LIN {X 0,Y 497.703,Z 599.514,A -85,B 0,C 180,E1 23826.812,E2 23826.812} C_VEL
LIN {X 0,Y 498.495,Z 582.352,A -85,B 0,C 180,E1 23826.005,E2 23826.005} C_VEL
LIN {X 0,Y 499.076,Z 563.889,A -85,B 0,C 180,E1 23825.37,E2 23825.37} C_VEL
LIN {X 0,Y 499.352,Z 545.212,A -85,B 0,C 180,E1 23824.95,E2 23824.95} C_VEL
LIN {X 0,Y 500.791,Z 353.157,A -85,B 0,C 180,E1 23822.188,E2 23822.188} C_VEL
LIN {X 0,Y 497.596,Z 338.367,A -85,B 0,C 180,E1 23821.709,E2 23821.709} C_VEL
LIN {X 0,Y 497.97,Z 328.618,A -85,B 0,C 180,E1 23820.732,E2 23820.732} C_VEL
LIN {X 0,Y 491.564,Z 309.601,A -85,B 0,C 180,E1 23818.115,E2 23818.115} C_VEL
LIN {X 0,Y 488.836,Z 301.801,A -85,B 0,C 180,E1 23816.953,E2 23816.953} C_VEL
LIN {X 0,Y 488.821,Z 301.599,A -85,B 0,C 180,E1 23813.618,E2 23813.618} C_VEL
LIN {X 0,Y 488.832,Z 301.582,A -85,B 0,C 180,E1 23810.041,E2 23810.041} C_VEL
LIN {X 0,Y 488.806,Z 301.568,A -85,B 0,C 180,E1 23806.566,E2 23806.566} C_VEL
LIN {X 0,Y 488.795,Z 301.598,A -85,B 0,C 180,E1 23803.093,E2 23803.093} C_VEL
LIN {X 0,Y 488.83,Z 301.598,A -85,B 0,C 180,E1 23799.656,E2 23799.656} C_VEL
LIN {X 0,Y 488.827,Z 301.593,A -85,B 0,C 180,E1 23796.092,E2 23796.092} C_VEL
LIN {X 0,Y 488.788,Z 301.595,A -85,B 0,C 180,E1 23792.568,E2 23792.568} C_VEL
LIN {X 0,Y 488.784,Z 301.593,A -85,B 0,C 180,E1 23789,E2 23789} C_VEL
LIN {X 0,Y 488.822,Z 301.587,A -85,B 0,C 180,E1 23785.569,E2 23785.569} C_VEL
LIN {X 0,Y 488.805,Z 301.596,A -85,B 0,C 180,E1 23782.09,E2 23782.09} C_VEL
LIN {X 0,Y 488.769,Z 301.592,A -85,B 0,C 180,E1 23778.61,E2 23778.61} C_VEL
LIN {X 0,Y 488.776,Z 301.588,A -85,B 0,C 180,E1 23775.058,E2 23775.058} C_VEL
LIN {X 0,Y 488.818,Z 301.596,A -85,B 0,C 180,E1 23771.684,E2 23771.684} C_VEL
LIN {X 0,Y 488.765,Z 301.585,A -85,B 0,C 180,E1 23768.233,E2 23768.233} C_VEL
LIN {X 0,Y 488.755,Z 301.597,A -85,B 0,C 180,E1 23764.694,E2 23764.694} C_VEL
LIN {X 0,Y 488.797,Z 301.596,A -85,B 0,C 180,E1 23761.29,E2 23761.29} C_VEL
LIN {X 0,Y 488.775,Z 301.592,A -85,B 0,C 180,E1 23757.89,E2 23757.89} C_VEL
LIN {X 0,Y 488.754,Z 301.599,A -85,B 0,C 180,E1 23754.483,E2 23754.483} C_VEL
LIN {X 0,Y 488.789,Z 301.592,A -85,B 0,C 180,E1 23751.057,E2 23751.057} C_VEL
LIN {X 0,Y 488.805,Z 301.592,A -85,B 0,C 180,E1 23747.598,E2 23747.598} C_VEL
LIN {X 0,Y 488.767,Z 301.599,A -85,B 0,C 180,E1 23744.212,E2 23744.212} C_VEL
LIN {X 0,Y 488.78,Z 301.595,A -85,B 0,C 180,E1 23740.647,E2 23740.647} C_VEL
LIN {X 0,Y 488.836,Z 301.585,A -85,B 0,C 180,E1 23737.258,E2 23737.258} C_VEL
LIN {X 0,Y 488.792,Z 301.599,A -85,B 0,C 180,E1 23733.779,E2 23733.779} C_VEL
LIN {X 0,Y 488.782,Z 301.597,A -85,B 0,C 180,E1 23730.328,E2 23730.328} C_VEL
LIN {X 0,Y 488.822,Z 301.594,A -85,B 0,C 180,E1 23726.898,E2 23726.898} C_VEL
LIN {X 0,Y 488.826,Z 301.564,A -85,B 0,C 180,E1 23723.301,E2 23723.301} C_VEL
LIN {X 0,Y 488.793,Z 301.59,A -85,B 0,C 180,E1 23719.883,E2 23719.883} C_VEL
LIN {X 0,Y 488.796,Z 301.598,A -85,B 0,C 180,E1 23716.225,E2 23716.225} C_VEL
LIN {X 0,Y 488.826,Z 301.575,A -85,B 0,C 180,E1 23712.751,E2 23712.751} C_VEL
LIN {X 0,Y 488.839,Z 301.65,A -85,B 0,C 180,E1 23711.1,E2 23711.1} C_VEL
LIN {X 0,Y 489.193,Z 303.151,A -85,B 0,C 180,E1 23710.866,E2 23710.866} C_VEL
LIN {X 0,Y 497.247,Z 321.838,A -85,B 0,C 180,E1 23708.815,E2 23708.815} C_VEL
LIN {X 0,Y 502.538,Z 335.639,A -85,B 0,C 180,E1 23707.431,E2 23707.431} C_VEL
LIN {X 0,Y 500.242,Z 388.267,A -85,B 0,C 180,E1 23704.007,E2 23704.007} C_VEL
LIN {X 0,Y 502.743,Z 409.204,A -85,B 0,C 180,E1 23703.487,E2 23703.487} C_VEL
LIN {X 0,Y 499.827,Z 627.706,A -85,B 0,C 180,E1 23700.075,E2 23700.075} C_VEL
LIN {X 0,Y 499.277,Z 655.552,A -85,B 0,C 180,E1 23699.579,E2 23699.579} C_VEL
LIN {X 0,Y 498.434,Z 677.22,A -85,B 0,C 180,E1 23698.977,E2 23698.977} C_VEL
LIN {X 0,Y 497.483,Z 697.861,A -85,B 0,C 180,E1 23698.184,E2 23698.184} C_VEL
LIN {X 0,Y 496.413,Z 717.588,A -85,B 0,C 180,E1 23697.207,E2 23697.207} C_VEL
LIN {X 0,Y 495.194,Z 737.474,A -85,B 0,C 180,E1 23695.985,E2 23695.985} C_VEL
LIN {X 0,Y 493.989,Z 756.462,A -85,B 0,C 180,E1 23694.565,E2 23694.565} C_VEL
LIN {X 0,Y 492.797,Z 774.049,A -85,B 0,C 180,E1 23692.989,E2 23692.989} C_VEL
LIN {X 0,Y 491.739,Z 789.65,A -85,B 0,C 180,E1 23691.343,E2 23691.343} C_VEL
LIN {X 0,Y 490.759,Z 804.438,A -85,B 0,C 180,E1 23689.519,E2 23689.519} C_VEL
LIN {X 0,Y 490.048,Z 815.118,A -85,B 0,C 180,E1 23687.944,E2 23687.944} C_VEL
LIN {X 0,Y 489.28,Z 826.646,A -85,B 0,C 180,E1 23685.892,E2 23685.892} C_VEL
LIN {X 0,Y 488.709,Z 836.846,A -85,B 0,C 180,E1 23683.728,E2 23683.728} C_VEL
LIN {X 0,Y 488.31,Z 845.655,A -85,B 0,C 180,E1 23681.456,E2 23681.456} C_VEL
LIN {X 0,Y 488.088,Z 852.685,A -85,B 0,C 180,E1 23679.194,E2 23679.194} C_VEL
LIN {X 0,Y 487.97,Z 858.26,A -85,B 0,C 180,E1 23676.825,E2 23676.825} C_VEL
LIN {X 0,Y 487.913,Z 862.087,A -85,B 0,C 180,E1 23674.466,E2 23674.466} C_VEL
LIN {X 0,Y 487.908,Z 864.304,A -85,B 0,C 180,E1 23672.114,E2 23672.114} C_VEL
LIN {X 0,Y 487.906,Z 864.962,A -85,B 0,C 180,E1 23669.765,E2 23669.765} C_VEL
LIN {X 0,Y 487.905,Z 864.03,A -85,B 0,C 180,E1 23667.416,E2 23667.416} C_VEL
LIN {X 0,Y 487.929,Z 861.446,A -85,B 0,C 180,E1 23665.063,E2 23665.063} C_VEL
LIN {X 0,Y 487.987,Z 857.244,A -85,B 0,C 180,E1 23662.702,E2 23662.702} C_VEL
LIN {X 0,Y 488.126,Z 851.326,A -85,B 0,C 180,E1 23660.331,E2 23660.331} C_VEL
LIN {X 0,Y 488.381,Z 844.01,A -85,B 0,C 180,E1 23658.067,E2 23658.067} C_VEL
LIN {X 0,Y 488.823,Z 834.789,A -85,B 0,C 180,E1 23655.792,E2 23655.792} C_VEL
LIN {X 0,Y 489.44,Z 824.106,A -85,B 0,C 180,E1 23653.626,E2 23653.626} C_VEL
LIN {X 0,Y 490.253,Z 812.019,A -85,B 0,C 180,E1 23651.572,E2 23651.572} C_VEL
LIN {X 0,Y 491.025,Z 800.468,A -85,B 0,C 180,E1 23649.954,E2 23649.954} C_VEL
LIN {X 0,Y 492.085,Z 784.784,A -85,B 0,C 180,E1 23648.109,E2 23648.109} C_VEL
LIN {X 0,Y 493.241,Z 767.415,A -85,B 0,C 180,E1 23646.385,E2 23646.385} C_VEL
LIN {X 0,Y 494.4,Z 750.145,A -85,B 0,C 180,E1 23644.94,E2 23644.94} C_VEL
LIN {X 0,Y 495.552,Z 731.825,A -85,B 0,C 180,E1 23643.649,E2 23643.649} C_VEL
LIN {X 0,Y 496.728,Z 711.811,A -85,B 0,C 180,E1 23642.487,E2 23642.487} C_VEL
LIN {X 0,Y 497.765,Z 692.146,A -85,B 0,C 180,E1 23641.572,E2 23641.572} C_VEL
LIN {X 0,Y 498.696,Z 671.504,A -85,B 0,C 180,E1 23640.837,E2 23640.837} C_VEL
LIN {X 0,Y 499.453,Z 649.882,A -85,B 0,C 180,E1 23640.293,E2 23640.293} C_VEL
LIN {X 0,Y 502.656,Z 414.695,A -85,B 0,C 180,E1 23636.6,E2 23636.6} C_VEL
LIN {X 0,Y 502.523,Z 405.875,A -85,B 0,C 180,E1 23636.443,E2 23636.443} C_VEL
LIN {X 0,Y 500.189,Z 387.515,A -85,B 0,C 180,E1 23635.965,E2 23635.965} C_VEL
LIN {X 0,Y 502.552,Z 335.273,A -85,B 0,C 180,E1 23632.545,E2 23632.545} C_VEL
LIN {X 0,Y 494.184,Z 314.542,A -85,B 0,C 180,E1 23630.409,E2 23630.409} C_VEL
LIN {X 0,Y 488.897,Z 302.02,A -85,B 0,C 180,E1 23628.995,E2 23628.995} C_VEL
LIN {X 0,Y 488.827,Z 301.588,A -85,B 0,C 180,E1 23628.648,E2 23628.648} C_VEL
LIN {X 0,Y 488.832,Z 301.584,A -85,B 0,C 180,E1 23625.049,E2 23625.049} C_VEL
LIN {X 0,Y 488.802,Z 301.566,A -85,B 0,C 180,E1 23621.51,E2 23621.51} C_VEL
LIN {X 0,Y 488.79,Z 301.592,A -85,B 0,C 180,E1 23618.004,E2 23618.004} C_VEL
LIN {X 0,Y 488.813,Z 301.58,A -85,B 0,C 180,E1 23614.482,E2 23614.482} C_VEL
LIN {X 0,Y 488.834,Z 301.587,A -85,B 0,C 180,E1 23610.89,E2 23610.89} C_VEL
LIN {X 0,Y 488.79,Z 301.591,A -85,B 0,C 180,E1 23607.403,E2 23607.403} C_VEL
LIN {X 0,Y 488.779,Z 301.593,A -85,B 0,C 180,E1 23603.884,E2 23603.884} C_VEL
LIN {X 0,Y 488.816,Z 301.598,A -85,B 0,C 180,E1 23600.473,E2 23600.473} C_VEL
LIN {X 0,Y 488.801,Z 301.592,A -85,B 0,C 180,E1 23597.008,E2 23597.008} C_VEL
LIN {X 0,Y 488.765,Z 301.585,A -85,B 0,C 180,E1 23593.606,E2 23593.606} C_VEL
LIN {X 0,Y 488.783,Z 301.596,A -85,B 0,C 180,E1 23590.132,E2 23590.132} C_VEL
LIN {X 0,Y 488.827,Z 301.591,A -85,B 0,C 180,E1 23586.577,E2 23586.577} C_VEL
LIN {X 0,Y 488.77,Z 301.59,A -85,B 0,C 180,E1 23583.049,E2 23583.049} C_VEL
LIN {X 0,Y 488.753,Z 301.6,A -85,B 0,C 180,E1 23579.648,E2 23579.648} C_VEL
LIN {X 0,Y 488.794,Z 301.59,A -85,B 0,C 180,E1 23576.247,E2 23576.247} C_VEL
LIN {X 0,Y 488.783,Z 301.599,A -85,B 0,C 180,E1 23572.79,E2 23572.79} C_VEL
LIN {X 0,Y 488.756,Z 301.598,A -85,B 0,C 180,E1 23569.39,E2 23569.39} C_VEL
LIN {X 0,Y 488.783,Z 301.585,A -85,B 0,C 180,E1 23565.911,E2 23565.911} C_VEL
LIN {X 0,Y 488.808,Z 301.6,A -85,B 0,C 180,E1 23562.501,E2 23562.501} C_VEL
LIN {X 0,Y 488.771,Z 301.593,A -85,B 0,C 180,E1 23559.023,E2 23559.023} C_VEL
LIN {X 0,Y 488.775,Z 301.586,A -85,B 0,C 180,E1 23555.464,E2 23555.464} C_VEL
LIN {X 0,Y 488.83,Z 301.592,A -85,B 0,C 180,E1 23552.069,E2 23552.069} C_VEL
LIN {X 0,Y 488.806,Z 301.597,A -85,B 0,C 180,E1 23548.534,E2 23548.534} C_VEL
LIN {X 0,Y 488.781,Z 301.595,A -85,B 0,C 180,E1 23545.056,E2 23545.056} C_VEL
LIN {X 0,Y 488.801,Z 301.594,A -85,B 0,C 180,E1 23541.549,E2 23541.549} C_VEL
LIN {X 0,Y 488.832,Z 301.59,A -85,B 0,C 180,E1 23538.022,E2 23538.022} C_VEL
LIN {X 0,Y 488.81,Z 301.571,A -85,B 0,C 180,E1 23534.448,E2 23534.448} C_VEL
LIN {X 0,Y 488.793,Z 301.6,A -85,B 0,C 180,E1 23530.887,E2 23530.887} C_VEL
LIN {X 0,Y 488.804,Z 301.585,A -85,B 0,C 180,E1 23527.277,E2 23527.277} C_VEL
LIN {X 0,Y 488.829,Z 301.571,A -85,B 0,C 180,E1 23523.803,E2 23523.803} C_VEL
LIN {X 0,Y 488.825,Z 301.575,A -85,B 0,C 180,E1 23523.535,E2 23523.535} C_VEL
LIN {X 0,Y 488.707,Z 302.659,A -85,B 0,C 180,E1 23523.028,E2 23523.028} C_VEL
LIN {X 0,Y 488.366,Z 306.029,A -85,B 0,C 180,E1 23522.479,E2 23522.479} C_VEL
LIN {X 0,Y 487.643,Z 319.511,A -85,B 0,C 180,E1 23521.022,E2 23521.022} C_VEL
LIN {X 0,Y 488.549,Z 324.711,A -85,B 0,C 180,E1 23520.361,E2 23520.361} C_VEL
LIN {X 0,Y 490.865,Z 331.872,A -85,B 0,C 180,E1 23519.399,E2 23519.399} C_VEL
LIN {X 0,Y 490.606,Z 339.583,A -85,B 0,C 180,E1 23518.658,E2 23518.658} C_VEL
LIN {X 0,Y 494.065,Z 356.306,A -85,B 0,C 180,E1 23518.141,E2 23518.141} C_VEL
LIN {X 0,Y 492.291,Z 551.901,A -85,B 0,C 180,E1 23515.29,E2 23515.29} C_VEL
LIN {X 0,Y 491.896,Z 570.892,A -85,B 0,C 180,E1 23514.786,E2 23514.786} C_VEL
LIN {X 0,Y 491.192,Z 588.904,A -85,B 0,C 180,E1 23514.087,E2 23514.087} C_VEL
LIN {X 0,Y 490.248,Z 606.351,A -85,B 0,C 180,E1 23513.179,E2 23513.179} C_VEL
LIN {X 0,Y 489.098,Z 622.756,A -85,B 0,C 180,E1 23512.095,E2 23512.095} C_VEL
LIN {X 0,Y 487.851,Z 638.101,A -85,B 0,C 180,E1 23510.839,E2 23510.839} C_VEL
LIN {X 0,Y 486.5,Z 652.717,A -85,B 0,C 180,E1 23509.379,E2 23509.379} C_VEL
LIN {X 0,Y 485.184,Z 666.107,A -85,B 0,C 180,E1 23507.757,E2 23507.757} C_VEL
LIN {X 0,Y 483.924,Z 678.429,A -85,B 0,C 180,E1 23505.949,E2 23505.949} C_VEL
LIN {X 0,Y 482.864,Z 689.222,A -85,B 0,C 180,E1 23504.02,E2 23504.02} C_VEL
LIN {X 0,Y 481.974,Z 698.544,A -85,B 0,C 180,E1 23501.973,E2 23501.973} C_VEL
LIN {X 0,Y 481.314,Z 706.381,A -85,B 0,C 180,E1 23499.807,E2 23499.807} C_VEL
LIN {X 0,Y 480.863,Z 712.699,A -85,B 0,C 180,E1 23497.527,E2 23497.527} C_VEL
LIN {X 0,Y 480.577,Z 717.234,A -85,B 0,C 180,E1 23495.252,E2 23495.252} C_VEL
LIN {X 0,Y 480.428,Z 720.208,A -85,B 0,C 180,E1 23492.863,E2 23492.863} C_VEL
LIN {X 0,Y 480.381,Z 721.437,A -85,B 0,C 180,E1 23490.477,E2 23490.477} C_VEL
LIN {X 0,Y 480.403,Z 720.959,A -85,B 0,C 180,E1 23488.092,E2 23488.092} C_VEL
LIN {X 0,Y 480.492,Z 718.906,A -85,B 0,C 180,E1 23485.824,E2 23485.824} C_VEL
LIN {X 0,Y 480.694,Z 715.237,A -85,B 0,C 180,E1 23483.551,E2 23483.551} C_VEL
LIN {X 0,Y 481.06,Z 709.851,A -85,B 0,C 180,E1 23481.273,E2 23481.273} C_VEL
LIN {X 0,Y 481.58,Z 703.016,A -85,B 0,C 180,E1 23479.11,E2 23479.11} C_VEL
LIN {X 0,Y 482.32,Z 694.791,A -85,B 0,C 180,E1 23477.063,E2 23477.063} C_VEL
LIN {X 0,Y 483.286,Z 684.793,A -85,B 0,C 180,E1 23475.054,E2 23475.054} C_VEL
LIN {X 0,Y 484.416,Z 673.543,A -85,B 0,C 180,E1 23473.204,E2 23473.204} C_VEL
LIN {X 0,Y 485.68,Z 661.12,A -85,B 0,C 180,E1 23471.517,E2 23471.517} C_VEL
LIN {X 0,Y 487.013,Z 647.199,A -85,B 0,C 180,E1 23469.95,E2 23469.95} C_VEL
LIN {X 0,Y 488.338,Z 632.237,A -85,B 0,C 180,E1 23468.564,E2 23468.564} C_VEL
LIN {X 0,Y 489.56,Z 616.352,A -85,B 0,C 180,E1 23467.364,E2 23467.364} C_VEL
LIN {X 0,Y 490.6,Z 600.329,A -85,B 0,C 180,E1 23466.393,E2 23466.393} C_VEL
LIN {X 0,Y 491.444,Z 583.063,A -85,B 0,C 180,E1 23465.575,E2 23465.575} C_VEL
LIN {X 0,Y 492.049,Z 564.71,A -85,B 0,C 180,E1 23464.938,E2 23464.938} C_VEL
LIN {X 0,Y 492.337,Z 545.999,A -85,B 0,C 180,E1 23464.513,E2 23464.513} C_VEL
LIN {X 0,Y 493.96,Z 354.759,A -85,B 0,C 180,E1 23461.732,E2 23461.732} C_VEL
LIN {X 0,Y 490.529,Z 338.771,A -85,B 0,C 180,E1 23461.202,E2 23461.202} C_VEL
LIN {X 0,Y 490.727,Z 331.435,A -85,B 0,C 180,E1 23460.458,E2 23460.458} C_VEL
LIN {X 0,Y 484.023,Z 311.463,A -85,B 0,C 180,E1 23457.66,E2 23457.66} C_VEL
LIN {X 0,Y 480.917,Z 302.763,A -85,B 0,C 180,E1 23456.336,E2 23456.336} C_VEL
LIN {X 0,Y 480.867,Z 302.575,A -85,B 0,C 180,E1 23452.767,E2 23452.767} C_VEL
LIN {X 0,Y 480.863,Z 302.589,A -85,B 0,C 180,E1 23449.189,E2 23449.189} C_VEL
LIN {X 0,Y 480.883,Z 302.553,A -85,B 0,C 180,E1 23445.664,E2 23445.664} C_VEL
LIN {X 0,Y 480.895,Z 302.58,A -85,B 0,C 180,E1 23442.028,E2 23442.028} C_VEL
LIN {X 0,Y 480.867,Z 302.582,A -85,B 0,C 180,E1 23438.441,E2 23438.441} C_VEL
LIN {X 0,Y 480.848,Z 302.582,A -85,B 0,C 180,E1 23434.878,E2 23434.878} C_VEL
LIN {X 0,Y 480.86,Z 302.585,A -85,B 0,C 180,E1 23431.288,E2 23431.288} C_VEL
LIN {X 0,Y 480.894,Z 302.581,A -85,B 0,C 180,E1 23427.758,E2 23427.758} C_VEL
LIN {X 0,Y 480.86,Z 302.573,A -85,B 0,C 180,E1 23424.182,E2 23424.182} C_VEL
LIN {X 0,Y 480.835,Z 302.581,A -85,B 0,C 180,E1 23420.657,E2 23420.657} C_VEL
LIN {X 0,Y 480.84,Z 302.588,A -85,B 0,C 180,E1 23417.05,E2 23417.05} C_VEL
LIN {X 0,Y 480.885,Z 302.571,A -85,B 0,C 180,E1 23413.589,E2 23413.589} C_VEL
LIN {X 0,Y 480.844,Z 302.586,A -85,B 0,C 180,E1 23410.06,E2 23410.06} C_VEL
LIN {X 0,Y 480.818,Z 302.588,A -85,B 0,C 180,E1 23406.568,E2 23406.568} C_VEL
LIN {X 0,Y 480.836,Z 302.574,A -85,B 0,C 180,E1 23403.099,E2 23403.099} C_VEL
LIN {X 0,Y 480.876,Z 302.585,A -85,B 0,C 180,E1 23399.524,E2 23399.524} C_VEL
LIN {X 0,Y 480.831,Z 302.58,A -85,B 0,C 180,E1 23395.946,E2 23395.946} C_VEL
LIN {X 0,Y 480.818,Z 302.579,A -85,B 0,C 180,E1 23392.472,E2 23392.472} C_VEL
LIN {X 0,Y 480.845,Z 302.587,A -85,B 0,C 180,E1 23388.943,E2 23388.943} C_VEL
LIN {X 0,Y 480.886,Z 302.576,A -85,B 0,C 180,E1 23385.429,E2 23385.429} C_VEL
LIN {X 0,Y 480.839,Z 302.581,A -85,B 0,C 180,E1 23381.951,E2 23381.951} C_VEL
LIN {X 0,Y 480.834,Z 302.586,A -85,B 0,C 180,E1 23378.353,E2 23378.353} C_VEL
LIN {X 0,Y 480.87,Z 302.585,A -85,B 0,C 180,E1 23374.902,E2 23374.902} C_VEL
LIN {X 0,Y 480.897,Z 302.584,A -85,B 0,C 180,E1 23371.296,E2 23371.296} C_VEL
LIN {X 0,Y 480.853,Z 302.585,A -85,B 0,C 180,E1 23367.808,E2 23367.808} C_VEL
LIN {X 0,Y 480.845,Z 302.554,A -85,B 0,C 180,E1 23364.187,E2 23364.187} C_VEL
LIN {X 0,Y 480.874,Z 302.584,A -85,B 0,C 180,E1 23360.642,E2 23360.642} C_VEL
LIN {X 0,Y 480.892,Z 302.564,A -85,B 0,C 180,E1 23357.041,E2 23357.041} C_VEL
LIN {X 0,Y 480.874,Z 302.557,A -85,B 0,C 180,E1 23353.477,E2 23353.477} C_VEL
LIN {X 0,Y 480.906,Z 302.863,A -85,B 0,C 180,E1 23351.68,E2 23351.68} C_VEL
LIN {X 0,Y 483.793,Z 309.643,A -85,B 0,C 180,E1 23350.851,E2 23350.851} C_VEL
LIN {X 0,Y 493.151,Z 332.06,A -85,B 0,C 180,E1 23348.407,E2 23348.407} C_VEL
LIN {X 0,Y 495.521,Z 338.509,A -85,B 0,C 180,E1 23347.762,E2 23347.762} C_VEL
LIN {X 0,Y 493.157,Z 387.828,A -85,B 0,C 180,E1 23344.503,E2 23344.503} C_VEL
LIN {X 0,Y 495.787,Z 410.337,A -85,B 0,C 180,E1 23343.929,E2 23343.929} C_VEL
LIN {X 0,Y 492.138,Z 649.298,A -85,B 0,C 180,E1 23340.091,E2 23340.091} C_VEL
LIN {X 0,Y 491.304,Z 671.237,A -85,B 0,C 180,E1 23339.525,E2 23339.525} C_VEL
LIN {X 0,Y 490.246,Z 692.612,A -85,B 0,C 180,E1 23338.74,E2 23338.74} C_VEL
LIN {X 0,Y 489.065,Z 713.265,A -85,B 0,C 180,E1 23337.746,E2 23337.746} C_VEL
LIN {X 0,Y 487.862,Z 732.316,A -85,B 0,C 180,E1 23336.602,E2 23336.602} C_VEL
LIN {X 0,Y 486.592,Z 751.078,A -85,B 0,C 180,E1 23335.237,E2 23335.237} C_VEL
LIN {X 0,Y 485.262,Z 769.522,A -85,B 0,C 180,E1 23333.625,E2 23333.625} C_VEL
LIN {X 0,Y 484.067,Z 786.361,A -85,B 0,C 180,E1 23331.874,E2 23331.874} C_VEL
LIN {X 0,Y 483.041,Z 800.956,A -85,B 0,C 180,E1 23330.096,E2 23330.096} C_VEL
LIN {X 0,Y 482.123,Z 814.745,A -85,B 0,C 180,E1 23328.124,E2 23328.124} C_VEL
LIN {X 0,Y 481.36,Z 827.01,A -85,B 0,C 180,E1 23326.037,E2 23326.037} C_VEL
LIN {X 0,Y 480.828,Z 836.331,A -85,B 0,C 180,E1 23324.081,E2 23324.081} C_VEL
LIN {X 0,Y 480.378,Z 845.25,A -85,B 0,C 180,E1 23321.769,E2 23321.769} C_VEL
LIN {X 0,Y 480.123,Z 852.375,A -85,B 0,C 180,E1 23319.469,E2 23319.469} C_VEL
LIN {X 0,Y 479.983,Z 858.006,A -85,B 0,C 180,E1 23317.059,E2 23317.059} C_VEL
LIN {X 0,Y 479.919,Z 861.926,A -85,B 0,C 180,E1 23314.66,E2 23314.66} C_VEL
LIN {X 0,Y 479.907,Z 864.303,A -85,B 0,C 180,E1 23312.149,E2 23312.149} C_VEL
LIN {X 0,Y 479.906,Z 864.962,A -85,B 0,C 180,E1 23309.761,E2 23309.761} C_VEL
LIN {X 0,Y 479.907,Z 864.03,A -85,B 0,C 180,E1 23307.373,E2 23307.373} C_VEL
LIN {X 0,Y 479.931,Z 861.445,A -85,B 0,C 180,E1 23304.98,E2 23304.98} C_VEL
LIN {X 0,Y 479.994,Z 857.159,A -85,B 0,C 180,E1 23302.54,E2 23302.54} C_VEL
LIN {X 0,Y 480.146,Z 851.326,A -85,B 0,C 180,E1 23300.168,E2 23300.168} C_VEL
LIN {X 0,Y 480.431,Z 844.009,A -85,B 0,C 180,E1 23297.866,E2 23297.866} C_VEL
LIN {X 0,Y 480.919,Z 834.786,A -85,B 0,C 180,E1 23295.553,E2 23295.553} C_VEL
LIN {X 0,Y 481.435,Z 825.653,A -85,B 0,C 180,E1 23293.718,E2 23293.718} C_VEL
LIN {X 0,Y 482.226,Z 813.101,A -85,B 0,C 180,E1 23291.63,E2 23291.63} C_VEL
LIN {X 0,Y 483.169,Z 799.084,A -85,B 0,C 180,E1 23289.657,E2 23289.657} C_VEL
LIN {X 0,Y 484.324,Z 782.977,A -85,B 0,C 180,E1 23287.741,E2 23287.741} C_VEL
LIN {X 0,Y 485.559,Z 765.638,A -85,B 0,C 180,E1 23286.004,E2 23286.004} C_VEL
LIN {X 0,Y 486.861,Z 747.174,A -85,B 0,C 180,E1 23284.452,E2 23284.452} C_VEL
LIN {X 0,Y 488.045,Z 729.442,A -85,B 0,C 180,E1 23283.211,E2 23283.211} C_VEL
LIN {X 0,Y 489.249,Z 710.207,A -85,B 0,C 180,E1 23282.096,E2 23282.096} C_VEL
LIN {X 0,Y 490.344,Z 690.339,A -85,B 0,C 180,E1 23281.169,E2 23281.169} C_VEL
LIN {X 0,Y 491.367,Z 669.669,A -85,B 0,C 180,E1 23280.429,E2 23280.429} C_VEL
LIN {X 0,Y 492.173,Z 648.273,A -85,B 0,C 180,E1 23279.887,E2 23279.887} C_VEL
LIN {X 0,Y 495.806,Z 409.537,A -85,B 0,C 180,E1 23276.057,E2 23276.057} C_VEL
LIN {X 0,Y 493.099,Z 386.873,A -85,B 0,C 180,E1 23275.46,E2 23275.46} C_VEL
LIN {X 0,Y 495.495,Z 338.18,A -85,B 0,C 180,E1 23272.214,E2 23272.214} C_VEL
LIN {X 0,Y 486.73,Z 316.473,A -85,B 0,C 180,E1 23269.925,E2 23269.925} C_VEL
LIN {X 0,Y 480.947,Z 303.081,A -85,B 0,C 180,E1 23268.366,E2 23268.366} C_VEL
LIN {X 0,Y 480.86,Z 302.587,A -85,B 0,C 180,E1 23268.107,E2 23268.107} C_VEL
LIN {X 0,Y 480.875,Z 302.584,A -85,B 0,C 180,E1 23264.483,E2 23264.483} C_VEL
LIN {X 0,Y 480.898,Z 302.556,A -85,B 0,C 180,E1 23260.818,E2 23260.818} C_VEL
LIN {X 0,Y 480.878,Z 302.561,A -85,B 0,C 180,E1 23257.22,E2 23257.22} C_VEL
LIN {X 0,Y 480.849,Z 302.585,A -85,B 0,C 180,E1 23253.724,E2 23253.724} C_VEL
LIN {X 0,Y 480.851,Z 302.589,A -85,B 0,C 180,E1 23250.074,E2 23250.074} C_VEL
LIN {X 0,Y 480.887,Z 302.578,A -85,B 0,C 180,E1 23246.616,E2 23246.616} C_VEL
LIN {X 0,Y 480.875,Z 302.576,A -85,B 0,C 180,E1 23243.01,E2 23243.01} C_VEL
LIN {X 0,Y 480.835,Z 302.584,A -85,B 0,C 180,E1 23239.559,E2 23239.559} C_VEL
LIN {X 0,Y 480.836,Z 302.588,A -85,B 0,C 180,E1 23235.931,E2 23235.931} C_VEL
LIN {X 0,Y 480.877,Z 302.576,A -85,B 0,C 180,E1 23232.488,E2 23232.488} C_VEL
LIN {X 0,Y 480.849,Z 302.58,A -85,B 0,C 180,E1 23228.972,E2 23228.972} C_VEL
LIN {X 0,Y 480.818,Z 302.589,A -85,B 0,C 180,E1 23225.489,E2 23225.489} C_VEL
LIN {X 0,Y 480.827,Z 302.584,A -85,B 0,C 180,E1 23221.906,E2 23221.906} C_VEL
LIN {X 0,Y 480.87,Z 302.579,A -85,B 0,C 180,E1 23218.451,E2 23218.451} C_VEL
LIN {X 0,Y 480.836,Z 302.586,A -85,B 0,C 180,E1 23214.87,E2 23214.87} C_VEL
LIN {X 0,Y 480.813,Z 302.574,A -85,B 0,C 180,E1 23211.389,E2 23211.389} C_VEL
LIN {X 0,Y 480.838,Z 302.586,A -85,B 0,C 180,E1 23207.876,E2 23207.876} C_VEL
LIN {X 0,Y 480.878,Z 302.577,A -85,B 0,C 180,E1 23204.441,E2 23204.441} C_VEL
LIN {X 0,Y 480.834,Z 302.582,A -85,B 0,C 180,E1 23200.945,E2 23200.945} C_VEL
LIN {X 0,Y 480.831,Z 302.587,A -85,B 0,C 180,E1 23197.375,E2 23197.375} C_VEL
LIN {X 0,Y 480.865,Z 302.585,A -85,B 0,C 180,E1 23193.844,E2 23193.844} C_VEL
LIN {X 0,Y 480.886,Z 302.575,A -85,B 0,C 180,E1 23190.34,E2 23190.34} C_VEL
LIN {X 0,Y 480.846,Z 302.586,A -85,B 0,C 180,E1 23186.847,E2 23186.847} C_VEL
LIN {X 0,Y 480.846,Z 302.586,A -85,B 0,C 180,E1 23183.181,E2 23183.181} C_VEL
LIN {X 0,Y 480.878,Z 302.582,A -85,B 0,C 180,E1 23179.711,E2 23179.711} C_VEL
LIN {X 0,Y 480.89,Z 302.58,A -85,B 0,C 180,E1 23176.175,E2 23176.175} C_VEL
LIN {X 0,Y 480.861,Z 302.567,A -85,B 0,C 180,E1 23172.601,E2 23172.601} C_VEL
LIN {X 0,Y 480.853,Z 302.564,A -85,B 0,C 180,E1 23169.052,E2 23169.052} C_VEL
LIN {X 0,Y 480.878,Z 302.572,A -85,B 0,C 180,E1 23165.457,E2 23165.457} C_VEL
LIN {X 0,Y 480.921,Z 302.801,A -85,B 0,C 180,E1 23163.554,E2 23163.554} C_VEL
LIN {X 0,Y 487.772,Z 322.317,A -85,B 0,C 180,E1 23160.69,E2 23160.69} C_VEL
LIN {X 0,Y 488.549,Z 324.711,A -85,B 0,C 180,E1 23160.361,E2 23160.361} C_VEL
LIN {X 0,Y 488.628,Z 327.991,A -85,B 0,C 180,E1 23159.994,E2 23159.994} C_VEL
LIN {X 0,Y 486.858,Z 333.513,A -85,B 0,C 180,E1 23159.555,E2 23159.555} C_VEL
LIN {X 0,Y 484.726,Z 340.308,A -85,B 0,C 180,E1 23159.192,E2 23159.192} C_VEL
LIN {X 0,Y 484.615,Z 344.653,A -85,B 0,C 180,E1 23159.02,E2 23159.02} C_VEL
LIN {X 0,Y 484.753,Z 345.376,A -85,B 0,C 180,E1 23158.995,E2 23158.995} C_VEL
LIN {X 0,Y 487.233,Z 357.819,A -85,B 0,C 180,E1 23158.611,E2 23158.611} C_VEL
LIN {X 0,Y 485.291,Z 552.929,A -85,B 0,C 180,E1 23155.73,E2 23155.73} C_VEL
LIN {X 0,Y 484.868,Z 571.912,A -85,B 0,C 180,E1 23155.219,E2 23155.219} C_VEL
LIN {X 0,Y 484.142,Z 589.615,A -85,B 0,C 180,E1 23154.525,E2 23154.525} C_VEL
LIN {X 0,Y 483.129,Z 607.284,A -85,B 0,C 180,E1 23153.597,E2 23153.597} C_VEL
LIN {X 0,Y 481.92,Z 623.618,A -85,B 0,C 180,E1 23152.506,E2 23152.506} C_VEL
LIN {X 0,Y 480.579,Z 639.115,A -85,B 0,C 180,E1 23151.223,E2 23151.223} C_VEL
LIN {X 0,Y 479.096,Z 654.161,A -85,B 0,C 180,E1 23149.696,E2 23149.696} C_VEL
LIN {X 0,Y 477.689,Z 667.548,A -85,B 0,C 180,E1 23148.046,E2 23148.046} C_VEL
LIN {X 0,Y 476.342,Z 679.831,A -85,B 0,C 180,E1 23146.21,E2 23146.21} C_VEL
LIN {X 0,Y 475.201,Z 690.591,A -85,B 0,C 180,E1 23144.251,E2 23144.251} C_VEL
LIN {X 0,Y 474.239,Z 699.883,A -85,B 0,C 180,E1 23142.171,E2 23142.171} C_VEL
LIN {X 0,Y 473.519,Z 707.693,A -85,B 0,C 180,E1 23139.971,E2 23139.971} C_VEL
LIN {X 0,Y 473.043,Z 713.704,A -85,B 0,C 180,E1 23137.774,E2 23137.774} C_VEL
LIN {X 0,Y 472.713,Z 718.291,A -85,B 0,C 180,E1 23135.462,E2 23135.462} C_VEL
LIN {X 0,Y 472.54,Z 721.219,A -85,B 0,C 180,E1 23133.154,E2 23133.154} C_VEL
LIN {X 0,Y 472.479,Z 722.598,A -85,B 0,C 180,E1 23130.728,E2 23130.728} C_VEL
LIN {X 0,Y 472.492,Z 722.289,A -85,B 0,C 180,E1 23128.302,E2 23128.302} C_VEL
LIN {X 0,Y 472.593,Z 720.28,A -85,B 0,C 180,E1 23125.875,E2 23125.875} C_VEL
LIN {X 0,Y 472.831,Z 716.498,A -85,B 0,C 180,E1 23123.443,E2 23123.443} C_VEL
LIN {X 0,Y 473.239,Z 711.145,A -85,B 0,C 180,E1 23121.128,E2 23121.128} C_VEL
LIN {X 0,Y 473.829,Z 704.179,A -85,B 0,C 180,E1 23118.882,E2 23118.882} C_VEL
LIN {X 0,Y 474.676,Z 695.612,A -85,B 0,C 180,E1 23116.727,E2 23116.727} C_VEL
LIN {X 0,Y 475.696,Z 685.842,A -85,B 0,C 180,E1 23114.747,E2 23114.747} C_VEL
LIN {X 0,Y 476.872,Z 674.958,A -85,B 0,C 180,E1 23112.931,E2 23112.931} C_VEL
LIN {X 0,Y 478.22,Z 662.576,A -85,B 0,C 180,E1 23111.218,E2 23111.218} C_VEL
LIN {X 0,Y 479.641,Z 648.71,A -85,B 0,C 180,E1 23109.628,E2 23109.628} C_VEL
LIN {X 0,Y 481.046,Z 633.823,A -85,B 0,C 180,E1 23108.223,E2 23108.223} C_VEL
LIN {X 0,Y 482.358,Z 617.867,A -85,B 0,C 180,E1 23106.994,E2 23106.994} C_VEL
LIN {X 0,Y 483.516,Z 601.071,A -85,B 0,C 180,E1 23105.961,E2 23105.961} C_VEL
LIN {X 0,Y 484.412,Z 583.702,A -85,B 0,C 180,E1 23105.131,E2 23105.131} C_VEL
LIN {X 0,Y 485.046,Z 565.341,A -85,B 0,C 180,E1 23104.49,E2 23104.49} C_VEL
LIN {X 0,Y 485.345,Z 546.648,A -85,B 0,C 180,E1 23104.064,E2 23104.064} C_VEL
LIN {X 0,Y 487.126,Z 356.194,A -85,B 0,C 180,E1 23101.259,E2 23101.259} C_VEL
LIN {X 0,Y 483.5,Z 339.269,A -85,B 0,C 180,E1 23100.687,E2 23100.687} C_VEL
LIN {X 0,Y 483.498,Z 334.249,A -85,B 0,C 180,E1 23100.171,E2 23100.171} C_VEL
LIN {X 0,Y 477.178,Z 315.408,A -85,B 0,C 180,E1 23097.499,E2 23097.499} C_VEL
LIN {X 0,Y 472.986,Z 303.82,A -85,B 0,C 180,E1 23095.72,E2 23095.72} C_VEL
LIN {X 0,Y 472.934,Z 303.576,A -85,B 0,C 180,E1 23093.403,E2 23093.403} C_VEL
LIN {X 0,Y 472.955,Z 303.563,A -85,B 0,C 180,E1 23089.746,E2 23089.746} C_VEL
LIN {X 0,Y 472.95,Z 303.537,A -85,B 0,C 180,E1 23086.1,E2 23086.1} C_VEL
LIN {X 0,Y 472.933,Z 303.573,A -85,B 0,C 180,E1 23082.454,E2 23082.454} C_VEL
LIN {X 0,Y 472.912,Z 303.573,A -85,B 0,C 180,E1 23078.898,E2 23078.898} C_VEL
LIN {X 0,Y 472.92,Z 303.573,A -85,B 0,C 180,E1 23075.253,E2 23075.253} C_VEL
LIN {X 0,Y 472.95,Z 303.576,A -85,B 0,C 180,E1 23071.621,E2 23071.621} C_VEL
LIN {X 0,Y 472.947,Z 303.568,A -85,B 0,C 180,E1 23067.991,E2 23067.991} C_VEL
LIN {X 0,Y 472.903,Z 303.562,A -85,B 0,C 180,E1 23064.482,E2 23064.482} C_VEL
LIN {X 0,Y 472.897,Z 303.57,A -85,B 0,C 180,E1 23060.852,E2 23060.852} C_VEL
LIN {X 0,Y 472.923,Z 303.577,A -85,B 0,C 180,E1 23057.344,E2 23057.344} C_VEL
LIN {X 0,Y 472.935,Z 303.558,A -85,B 0,C 180,E1 23053.822,E2 23053.822} C_VEL
LIN {X 0,Y 472.888,Z 303.575,A -85,B 0,C 180,E1 23050.354,E2 23050.354} C_VEL
LIN {X 0,Y 472.88,Z 303.577,A -85,B 0,C 180,E1 23046.678,E2 23046.678} C_VEL
LIN {X 0,Y 472.901,Z 303.562,A -85,B 0,C 180,E1 23043.152,E2 23043.152} C_VEL
LIN {X 0,Y 472.933,Z 303.575,A -85,B 0,C 180,E1 23039.555,E2 23039.555} C_VEL
LIN {X 0,Y 472.888,Z 303.569,A -85,B 0,C 180,E1 23035.999,E2 23035.999} C_VEL
LIN {X 0,Y 472.879,Z 303.568,A -85,B 0,C 180,E1 23032.467,E2 23032.467} C_VEL
LIN {X 0,Y 472.904,Z 303.576,A -85,B 0,C 180,E1 23028.907,E2 23028.907} C_VEL
LIN {X 0,Y 472.951,Z 303.566,A -85,B 0,C 180,E1 23025.304,E2 23025.304} C_VEL
LIN {X 0,Y 472.92,Z 303.565,A -85,B 0,C 180,E1 23021.67,E2 23021.67} C_VEL
LIN {X 0,Y 472.897,Z 303.575,A -85,B 0,C 180,E1 23018.15,E2 23018.15} C_VEL
LIN {X 0,Y 472.903,Z 303.575,A -85,B 0,C 180,E1 23014.449,E2 23014.449} C_VEL
LIN {X 0,Y 472.939,Z 303.574,A -85,B 0,C 180,E1 23010.906,E2 23010.906} C_VEL
LIN {X 0,Y 472.952,Z 303.576,A -85,B 0,C 180,E1 23007.286,E2 23007.286} C_VEL
LIN {X 0,Y 472.918,Z 303.538,A -85,B 0,C 180,E1 23003.702,E2 23003.702} C_VEL
LIN {X 0,Y 472.913,Z 303.572,A -85,B 0,C 180,E1 23000.126,E2 23000.126} C_VEL
LIN {X 0,Y 472.936,Z 303.564,A -85,B 0,C 180,E1 22996.599,E2 22996.599} C_VEL
LIN {X 0,Y 472.952,Z 303.545,A -85,B 0,C 180,E1 22992.99,E2 22992.99} C_VEL
LIN {X 0,Y 472.971,Z 303.857,A -85,B 0,C 180,E1 22992.351,E2 22992.351} C_VEL
LIN {X 0,Y 474.297,Z 307.162,A -85,B 0,C 180,E1 22991.914,E2 22991.914} C_VEL
LIN {X 0,Y 483.1,Z 327.539,A -85,B 0,C 180,E1 22989.561,E2 22989.561} C_VEL
LIN {X 0,Y 488.516,Z 341.444,A -85,B 0,C 180,E1 22988.097,E2 22988.097} C_VEL
LIN {X 0,Y 486.114,Z 387.432,A -85,B 0,C 180,E1 22985.012,E2 22985.012} C_VEL
LIN {X 0,Y 488.878,Z 411.471,A -85,B 0,C 180,E1 22984.387,E2 22984.387} C_VEL
LIN {X 0,Y 484.865,Z 648.353,A -85,B 0,C 180,E1 22980.495,E2 22980.495} C_VEL
LIN {X 0,Y 483.955,Z 670.357,A -85,B 0,C 180,E1 22979.916,E2 22979.916} C_VEL
LIN {X 0,Y 482.806,Z 691.638,A -85,B 0,C 180,E1 22979.121,E2 22979.121} C_VEL
LIN {X 0,Y 481.561,Z 712.103,A -85,B 0,C 180,E1 22978.119,E2 22978.119} C_VEL
LIN {X 0,Y 480.295,Z 730.708,A -85,B 0,C 180,E1 22976.988,E2 22976.988} C_VEL
LIN {X 0,Y 478.924,Z 749.74,A -85,B 0,C 180,E1 22975.592,E2 22975.592} C_VEL
LIN {X 0,Y 477.537,Z 768.213,A -85,B 0,C 180,E1 22973.965,E2 22973.965} C_VEL
LIN {X 0,Y 476.367,Z 783.896,A -85,B 0,C 180,E1 22972.327,E2 22972.327} C_VEL
LIN {X 0,Y 475.213,Z 799.277,A -85,B 0,C 180,E1 22970.442,E2 22970.442} C_VEL
LIN {X 0,Y 474.238,Z 813.225,A -85,B 0,C 180,E1 22968.422,E2 22968.422} C_VEL
LIN {X 0,Y 473.441,Z 825.496,A -85,B 0,C 180,E1 22966.312,E2 22966.312} C_VEL
LIN {X 0,Y 472.854,Z 835.853,A -85,B 0,C 180,E1 22964.198,E2 22964.198} C_VEL
LIN {X 0,Y 472.411,Z 844.926,A -85,B 0,C 180,E1 22961.971,E2 22961.971} C_VEL
LIN {X 0,Y 472.167,Z 851.3,A -85,B 0,C 180,E1 22959.999,E2 22959.999} C_VEL
LIN {X 0,Y 472.01,Z 856.987,A -85,B 0,C 180,E1 22957.669,E2 22957.669} C_VEL
LIN {X 0,Y 471.933,Z 861.287,A -85,B 0,C 180,E1 22955.227,E2 22955.227} C_VEL
LIN {X 0,Y 471.912,Z 863.954,A -85,B 0,C 180,E1 22952.793,E2 22952.793} C_VEL
LIN {X 0,Y 471.902,Z 864.939,A -85,B 0,C 180,E1 22950.364,E2 22950.364} C_VEL
LIN {X 0,Y 471.908,Z 864.37,A -85,B 0,C 180,E1 22947.936,E2 22947.936} C_VEL
LIN {X 0,Y 471.914,Z 862.243,A -85,B 0,C 180,E1 22945.504,E2 22945.504} C_VEL
LIN {X 0,Y 471.981,Z 858.51,A -85,B 0,C 180,E1 22943.065,E2 22943.065} C_VEL
LIN {X 0,Y 472.12,Z 852.991,A -85,B 0,C 180,E1 22940.615,E2 22940.615} C_VEL
LIN {X 0,Y 472.336,Z 846.662,A -85,B 0,C 180,E1 22938.523,E2 22938.523} C_VEL
LIN {X 0,Y 472.733,Z 838.068,A -85,B 0,C 180,E1 22936.298,E2 22936.298} C_VEL
LIN {X 0,Y 473.329,Z 827.515,A -85,B 0,C 180,E1 22934.062,E2 22934.062} C_VEL
LIN {X 0,Y 474.086,Z 815.458,A -85,B 0,C 180,E1 22931.94,E2 22931.94} C_VEL
LIN {X 0,Y 475.017,Z 802.008,A -85,B 0,C 180,E1 22929.935,E2 22929.935} C_VEL
LIN {X 0,Y 476.154,Z 786.614,A -85,B 0,C 180,E1 22927.987,E2 22927.987} C_VEL
LIN {X 0,Y 477.371,Z 770.423,A -85,B 0,C 180,E1 22926.248,E2 22926.248} C_VEL
LIN {X 0,Y 478.663,Z 753.619,A -85,B 0,C 180,E1 22924.719,E2 22924.719} C_VEL
LIN {X 0,Y 480.034,Z 734.524,A -85,B 0,C 180,E1 22923.263,E2 22923.263} C_VEL
LIN {X 0,Y 481.407,Z 714.406,A -85,B 0,C 180,E1 22922.006,E2 22922.006} C_VEL
LIN {X 0,Y 482.647,Z 694.418,A -85,B 0,C 180,E1 22921.004,E2 22921.004} C_VEL
LIN {X 0,Y 483.736,Z 674.042,A -85,B 0,C 180,E1 22920.21,E2 22920.21} C_VEL
LIN {X 0,Y 484.691,Z 652.903,A -85,B 0,C 180,E1 22919.611,E2 22919.611} C_VEL
LIN {X 0,Y 485.301,Z 625.97,A -85,B 0,C 180,E1 22919.119,E2 22919.119} C_VEL
LIN {X 0,Y 488.876,Z 409.615,A -85,B 0,C 180,E1 22915.579,E2 22915.579} C_VEL
LIN {X 0,Y 486.051,Z 386.321,A -85,B 0,C 180,E1 22914.944,E2 22914.944} C_VEL
LIN {X 0,Y 488.478,Z 341.211,A -85,B 0,C 180,E1 22911.885,E2 22911.885} C_VEL
LIN {X 0,Y 479.993,Z 320.207,A -85,B 0,C 180,E1 22909.623,E2 22909.623} C_VEL
LIN {X 0,Y 473.78,Z 306.31,A -85,B 0,C 180,E1 22907.975,E2 22907.975} C_VEL
LIN {X 0,Y 472.959,Z 303.774,A -85,B 0,C 180,E1 22907.625,E2 22907.625} C_VEL
LIN {X 0,Y 472.919,Z 303.578,A -85,B 0,C 180,E1 22904.073,E2 22904.073} C_VEL
LIN {X 0,Y 472.932,Z 303.554,A -85,B 0,C 180,E1 22900.441,E2 22900.441} C_VEL
LIN {X 0,Y 472.954,Z 303.54,A -85,B 0,C 180,E1 22896.898,E2 22896.898} C_VEL
LIN {X 0,Y 472.926,Z 303.572,A -85,B 0,C 180,E1 22893.346,E2 22893.346} C_VEL
LIN {X 0,Y 472.905,Z 303.577,A -85,B 0,C 180,E1 22889.792,E2 22889.792} C_VEL
LIN {X 0,Y 472.916,Z 303.575,A -85,B 0,C 180,E1 22886.223,E2 22886.223} C_VEL
LIN {X 0,Y 472.954,Z 303.563,A -85,B 0,C 180,E1 22882.629,E2 22882.629} C_VEL
LIN {X 0,Y 472.927,Z 303.567,A -85,B 0,C 180,E1 22879.001,E2 22879.001} C_VEL
LIN {X 0,Y 472.893,Z 303.576,A -85,B 0,C 180,E1 22875.45,E2 22875.45} C_VEL
LIN {X 0,Y 472.889,Z 303.576,A -85,B 0,C 180,E1 22871.785,E2 22871.785} C_VEL
LIN {X 0,Y 472.917,Z 303.563,A -85,B 0,C 180,E1 22868.266,E2 22868.266} C_VEL
LIN {X 0,Y 472.914,Z 303.577,A -85,B 0,C 180,E1 22864.851,E2 22864.851} C_VEL
LIN {X 0,Y 472.877,Z 303.573,A -85,B 0,C 180,E1 22861.332,E2 22861.332} C_VEL
LIN {X 0,Y 472.874,Z 303.566,A -85,B 0,C 180,E1 22857.697,E2 22857.697} C_VEL
LIN {X 0,Y 472.916,Z 303.577,A -85,B 0,C 180,E1 22854.175,E2 22854.175} C_VEL
LIN {X 0,Y 472.903,Z 303.561,A -85,B 0,C 180,E1 22850.753,E2 22850.753} C_VEL
LIN {X 0,Y 472.881,Z 303.575,A -85,B 0,C 180,E1 22847.297,E2 22847.297} C_VEL
LIN {X 0,Y 472.898,Z 303.576,A -85,B 0,C 180,E1 22843.714,E2 22843.714} C_VEL
LIN {X 0,Y 472.942,Z 303.56,A -85,B 0,C 180,E1 22840.179,E2 22840.179} C_VEL
LIN {X 0,Y 472.912,Z 303.577,A -85,B 0,C 180,E1 22836.711,E2 22836.711} C_VEL
LIN {X 0,Y 472.897,Z 303.576,A -85,B 0,C 180,E1 22833.153,E2 22833.153} C_VEL
LIN {X 0,Y 472.914,Z 303.572,A -85,B 0,C 180,E1 22829.608,E2 22829.608} C_VEL
LIN {X 0,Y 472.953,Z 303.563,A -85,B 0,C 180,E1 22826.074,E2 22826.074} C_VEL
LIN {X 0,Y 472.934,Z 303.568,A -85,B 0,C 180,E1 22822.447,E2 22822.447} C_VEL
LIN {X 0,Y 472.908,Z 303.573,A -85,B 0,C 180,E1 22819.006,E2 22819.006} C_VEL
LIN {X 0,Y 472.925,Z 303.565,A -85,B 0,C 180,E1 22815.419,E2 22815.419} C_VEL
LIN {X 0,Y 472.955,Z 303.563,A -85,B 0,C 180,E1 22811.913,E2 22811.913} C_VEL
LIN {X 0,Y 472.944,Z 303.544,A -85,B 0,C 180,E1 22808.274,E2 22808.274} C_VEL
LIN {X 0,Y 472.921,Z 303.549,A -85,B 0,C 180,E1 22804.66,E2 22804.66} C_VEL
LIN {X 0,Y 472.989,Z 303.849,A -85,B 0,C 180,E1 22804.174,E2 22804.174} C_VEL
LIN {X 0,Y 479.913,Z 323.35,A -85,B 0,C 180,E1 22801.249,E2 22801.249} C_VEL
LIN {X 0,Y 483.686,Z 335.439,A -85,B 0,C 180,E1 22799.606,E2 22799.606} C_VEL
LIN {X 0,Y 483.581,Z 340.099,A -85,B 0,C 180,E1 22799.172,E2 22799.172} C_VEL
LIN {X 0,Y 484.753,Z 345.376,A -85,B 0,C 180,E1 22798.995,E2 22798.995} C_VEL
LIN {X 0,Y 485.299,Z 350.755,A -85,B 0,C 180,E1 22798.868,E2 22798.868} C_VEL
LIN {X 0,Y 484.453,Z 358.492,A -85,B 0,C 180,E1 22798.806,E2 22798.806} C_VEL
LIN {X 0,Y 480.505,Z 376.325,A -85,B 0,C 180,E1 22798.815,E2 22798.815} C_VEL
LIN {X 0,Y 480.145,Z 380.86,A -85,B 0,C 180,E1 22798.769,E2 22798.769} C_VEL
LIN {X 0,Y 478.317,Z 553.703,A -85,B 0,C 180,E1 22796.188,E2 22796.188} C_VEL
LIN {X 0,Y 477.869,Z 572.764,A -85,B 0,C 180,E1 22795.669,E2 22795.669} C_VEL
LIN {X 0,Y 477.113,Z 590.257,A -85,B 0,C 180,E1 22794.977,E2 22794.977} C_VEL
LIN {X 0,Y 476.054,Z 607.893,A -85,B 0,C 180,E1 22794.045,E2 22794.045} C_VEL
LIN {X 0,Y 474.761,Z 624.43,A -85,B 0,C 180,E1 22792.93,E2 22792.93} C_VEL
LIN {X 0,Y 473.266,Z 640.634,A -85,B 0,C 180,E1 22791.567,E2 22791.567} C_VEL
LIN {X 0,Y 471.754,Z 655.085,A -85,B 0,C 180,E1 22790.081,E2 22790.081} C_VEL
LIN {X 0,Y 470.309,Z 668.075,A -85,B 0,C 180,E1 22788.467,E2 22788.467} C_VEL
LIN {X 0,Y 468.853,Z 680.476,A -85,B 0,C 180,E1 22786.604,E2 22786.604} C_VEL
LIN {X 0,Y 467.611,Z 691.334,A -85,B 0,C 180,E1 22784.614,E2 22784.614} C_VEL
LIN {X 0,Y 466.559,Z 700.713,A -85,B 0,C 180,E1 22782.5,E2 22782.5} C_VEL
LIN {X 0,Y 465.758,Z 708.599,A -85,B 0,C 180,E1 22780.263,E2 22780.263} C_VEL
LIN {X 0,Y 465.198,Z 714.956,A -85,B 0,C 180,E1 22777.906,E2 22777.906} C_VEL
LIN {X 0,Y 464.835,Z 719.52,A -85,B 0,C 180,E1 22775.554,E2 22775.554} C_VEL
LIN {X 0,Y 464.636,Z 722.483,A -85,B 0,C 180,E1 22773.143,E2 22773.143} C_VEL
LIN {X 0,Y 464.57,Z 723.8,A -85,B 0,C 180,E1 22770.74,E2 22770.74} C_VEL
LIN {X 0,Y 464.586,Z 723.493,A -85,B 0,C 180,E1 22768.273,E2 22768.273} C_VEL
LIN {X 0,Y 464.7,Z 721.497,A -85,B 0,C 180,E1 22765.805,E2 22765.805} C_VEL
LIN {X 0,Y 464.967,Z 717.736,A -85,B 0,C 180,E1 22763.332,E2 22763.332} C_VEL
LIN {X 0,Y 465.414,Z 712.406,A -85,B 0,C 180,E1 22760.977,E2 22760.977} C_VEL
LIN {X 0,Y 466.043,Z 705.625,A -85,B 0,C 180,E1 22758.742,E2 22758.742} C_VEL
LIN {X 0,Y 466.915,Z 697.454,A -85,B 0,C 180,E1 22756.628,E2 22756.628} C_VEL
LIN {X 0,Y 467.983,Z 687.949,A -85,B 0,C 180,E1 22754.638,E2 22754.638} C_VEL
LIN {X 0,Y 469.237,Z 677.125,A -85,B 0,C 180,E1 22752.772,E2 22752.772} C_VEL
LIN {X 0,Y 470.736,Z 664.265,A -85,B 0,C 180,E1 22750.944,E2 22750.944} C_VEL
LIN {X 0,Y 472.276,Z 650.183,A -85,B 0,C 180,E1 22749.296,E2 22749.296} C_VEL
LIN {X 0,Y 473.722,Z 635.791,A -85,B 0,C 180,E1 22747.907,E2 22747.907} C_VEL
LIN {X 0,Y 475.147,Z 619.6,A -85,B 0,C 180,E1 22746.631,E2 22746.631} C_VEL
LIN {X 0,Y 476.381,Z 602.871,A -85,B 0,C 180,E1 22745.577,E2 22745.577} C_VEL
LIN {X 0,Y 477.366,Z 585.014,A -85,B 0,C 180,E1 22744.705,E2 22744.705} C_VEL
LIN {X 0,Y 478.047,Z 566.621,A -85,B 0,C 180,E1 22744.051,E2 22744.051} C_VEL
LIN {X 0,Y 478.371,Z 547.772,A -85,B 0,C 180,E1 22743.611,E2 22743.611} C_VEL
LIN {X 0,Y 480.338,Z 357.695,A -85,B 0,C 180,E1 22740.775,E2 22740.775} C_VEL
LIN {X 0,Y 476.501,Z 339.597,A -85,B 0,C 180,E1 22740.144,E2 22740.144} C_VEL
LIN {X 0,Y 476.305,Z 337.122,A -85,B 0,C 180,E1 22739.868,E2 22739.868} C_VEL
LIN {X 0,Y 469.867,Z 318.049,A -85,B 0,C 180,E1 22737.138,E2 22737.138} C_VEL
LIN {X 0,Y 465.02,Z 304.778,A -85,B 0,C 180,E1 22735.041,E2 22735.041} C_VEL
LIN {X 0,Y 464.991,Z 304.532,A -85,B 0,C 180,E1 22731.423,E2 22731.423} C_VEL
LIN {X 0,Y 465.012,Z 304.548,A -85,B 0,C 180,E1 22727.868,E2 22727.868} C_VEL
LIN {X 0,Y 465.011,Z 304.552,A -85,B 0,C 180,E1 22724.16,E2 22724.16} C_VEL
LIN {X 0,Y 464.981,Z 304.56,A -85,B 0,C 180,E1 22720.62,E2 22720.62} C_VEL
LIN {X 0,Y 464.975,Z 304.563,A -85,B 0,C 180,E1 22717.021,E2 22717.021} C_VEL
LIN {X 0,Y 464.991,Z 304.555,A -85,B 0,C 180,E1 22713.4,E2 22713.4} C_VEL
LIN {X 0,Y 465.02,Z 304.55,A -85,B 0,C 180,E1 22709.781,E2 22709.781} C_VEL
LIN {X 0,Y 464.988,Z 304.563,A -85,B 0,C 180,E1 22706.156,E2 22706.156} C_VEL
LIN {X 0,Y 464.959,Z 304.565,A -85,B 0,C 180,E1 22702.639,E2 22702.639} C_VEL
LIN {X 0,Y 464.957,Z 304.557,A -85,B 0,C 180,E1 22698.949,E2 22698.949} C_VEL
LIN {X 0,Y 464.996,Z 304.553,A -85,B 0,C 180,E1 22695.464,E2 22695.464} C_VEL
LIN {X 0,Y 464.981,Z 304.562,A -85,B 0,C 180,E1 22691.914,E2 22691.914} C_VEL
LIN {X 0,Y 464.943,Z 304.549,A -85,B 0,C 180,E1 22688.409,E2 22688.409} C_VEL
LIN {X 0,Y 464.94,Z 304.564,A -85,B 0,C 180,E1 22684.688,E2 22684.688} C_VEL
LIN {X 0,Y 464.959,Z 304.567,A -85,B 0,C 180,E1 22681.109,E2 22681.109} C_VEL
LIN {X 0,Y 464.978,Z 304.55,A -85,B 0,C 180,E1 22677.659,E2 22677.659} C_VEL
LIN {X 0,Y 464.95,Z 304.566,A -85,B 0,C 180,E1 22674.075,E2 22674.075} C_VEL
LIN {X 0,Y 464.944,Z 304.562,A -85,B 0,C 180,E1 22670.469,E2 22670.469} C_VEL
LIN {X 0,Y 464.969,Z 304.549,A -85,B 0,C 180,E1 22666.929,E2 22666.929} C_VEL
LIN {X 0,Y 465.006,Z 304.561,A -85,B 0,C 180,E1 22663.383,E2 22663.383} C_VEL
LIN {X 0,Y 464.976,Z 304.563,A -85,B 0,C 180,E1 22659.745,E2 22659.745} C_VEL
LIN {X 0,Y 464.959,Z 304.558,A -85,B 0,C 180,E1 22656.289,E2 22656.289} C_VEL
LIN {X 0,Y 464.982,Z 304.554,A -85,B 0,C 180,E1 22652.741,E2 22652.741} C_VEL
LIN {X 0,Y 465.019,Z 304.552,A -85,B 0,C 180,E1 22649.221,E2 22649.221} C_VEL
LIN {X 0,Y 464.989,Z 304.544,A -85,B 0,C 180,E1 22645.562,E2 22645.562} C_VEL
LIN {X 0,Y 464.972,Z 304.556,A -85,B 0,C 180,E1 22642.048,E2 22642.048} C_VEL
LIN {X 0,Y 464.982,Z 304.528,A -85,B 0,C 180,E1 22638.442,E2 22638.442} C_VEL
LIN {X 0,Y 465.01,Z 304.541,A -85,B 0,C 180,E1 22634.801,E2 22634.801} C_VEL
LIN {X 0,Y 465.044,Z 304.759,A -85,B 0,C 180,E1 22633.079,E2 22633.079} C_VEL
LIN {X 0,Y 465.721,Z 306.981,A -85,B 0,C 180,E1 22632.757,E2 22632.757} C_VEL
LIN {X 0,Y 472.984,Z 323.119,A -85,B 0,C 180,E1 22630.782,E2 22630.782} C_VEL
LIN {X 0,Y 481.5,Z 344.299,A -85,B 0,C 180,E1 22628.449,E2 22628.449} C_VEL
LIN {X 0,Y 479.097,Z 386.938,A -85,B 0,C 180,E1 22625.539,E2 22625.539} C_VEL
LIN {X 0,Y 482.005,Z 412.581,A -85,B 0,C 180,E1 22624.859,E2 22624.859} C_VEL
LIN {X 0,Y 477.723,Z 644.596,A -85,B 0,C 180,E1 22620.972,E2 22620.972} C_VEL
LIN {X 0,Y 476.799,Z 665.677,A -85,B 0,C 180,E1 22620.435,E2 22620.435} C_VEL
LIN {X 0,Y 475.665,Z 685.998,A -85,B 0,C 180,E1 22619.705,E2 22619.705} C_VEL
LIN {X 0,Y 474.346,Z 706.844,A -85,B 0,C 180,E1 22618.723,E2 22618.723} C_VEL
LIN {X 0,Y 472.963,Z 726.232,A -85,B 0,C 180,E1 22617.578,E2 22617.578} C_VEL
LIN {X 0,Y 471.573,Z 744.752,A -85,B 0,C 180,E1 22616.251,E2 22616.251} C_VEL
LIN {X 0,Y 470.153,Z 762.824,A -85,B 0,C 180,E1 22614.701,E2 22614.701} C_VEL
LIN {X 0,Y 468.751,Z 780.33,A -85,B 0,C 180,E1 22612.909,E2 22612.909} C_VEL
LIN {X 0,Y 467.508,Z 796.111,A -85,B 0,C 180,E1 22610.991,E2 22610.991} C_VEL
LIN {X 0,Y 466.494,Z 809.868,A -85,B 0,C 180,E1 22609.013,E2 22609.013} C_VEL
LIN {X 0,Y 465.62,Z 822.611,A -85,B 0,C 180,E1 22606.851,E2 22606.851} C_VEL
LIN {X 0,Y 464.958,Z 833.863,A -85,B 0,C 180,E1 22604.572,E2 22604.572} C_VEL
LIN {X 0,Y 464.481,Z 843.122,A -85,B 0,C 180,E1 22602.304,E2 22602.304} C_VEL
LIN {X 0,Y 464.185,Z 850.907,A -85,B 0,C 180,E1 22599.922,E2 22599.922} C_VEL
LIN {X 0,Y 464.011,Z 856.844,A -85,B 0,C 180,E1 22597.553,E2 22597.553} C_VEL
LIN {X 0,Y 463.935,Z 861.3,A -85,B 0,C 180,E1 22595.069,E2 22595.069} C_VEL
LIN {X 0,Y 463.91,Z 863.893,A -85,B 0,C 180,E1 22592.718,E2 22592.718} C_VEL
LIN {X 0,Y 463.906,Z 864.873,A -85,B 0,C 180,E1 22590.247,E2 22590.247} C_VEL
LIN {X 0,Y 463.908,Z 864.253,A -85,B 0,C 180,E1 22587.9,E2 22587.9} C_VEL
LIN {X 0,Y 463.915,Z 862.156,A -85,B 0,C 180,E1 22585.55,E2 22585.55} C_VEL
LIN {X 0,Y 463.98,Z 858.403,A -85,B 0,C 180,E1 22583.193,E2 22583.193} C_VEL
LIN {X 0,Y 464.119,Z 852.952,A -85,B 0,C 180,E1 22580.827,E2 22580.827} C_VEL
LIN {X 0,Y 464.376,Z 845.677,A -85,B 0,C 180,E1 22578.426,E2 22578.426} C_VEL
LIN {X 0,Y 464.799,Z 836.645,A -85,B 0,C 180,E1 22576.059,E2 22576.059} C_VEL
LIN {X 0,Y 465.407,Z 826.027,A -85,B 0,C 180,E1 22573.783,E2 22573.783} C_VEL
LIN {X 0,Y 466.262,Z 813.125,A -85,B 0,C 180,E1 22571.496,E2 22571.496} C_VEL
LIN {X 0,Y 467.257,Z 799.418,A -85,B 0,C 180,E1 22569.456,E2 22569.456} C_VEL
LIN {X 0,Y 468.448,Z 784.198,A -85,B 0,C 180,E1 22567.539,E2 22567.539} C_VEL
LIN {X 0,Y 469.768,Z 767.411,A -85,B 0,C 180,E1 22565.747,E2 22565.747} C_VEL
LIN {X 0,Y 471.24,Z 748.867,A -85,B 0,C 180,E1 22564.083,E2 22564.083} C_VEL
LIN {X 0,Y 472.683,Z 730.027,A -85,B 0,C 180,E1 22562.675,E2 22562.675} C_VEL
LIN {X 0,Y 474.109,Z 710.405,A -85,B 0,C 180,E1 22561.468,E2 22561.468} C_VEL
LIN {X 0,Y 475.395,Z 690.615,A -85,B 0,C 180,E1 22560.484,E2 22560.484} C_VEL
LIN {X 0,Y 476.663,Z 668.946,A -85,B 0,C 180,E1 22559.663,E2 22559.663} C_VEL
LIN {X 0,Y 477.657,Z 646.844,A -85,B 0,C 180,E1 22559.072,E2 22559.072} C_VEL
LIN {X 0,Y 481.919,Z 417.222,A -85,B 0,C 180,E1 22555.218,E2 22555.218} C_VEL
LIN {X 0,Y 481.796,Z 409.235,A -85,B 0,C 180,E1 22555.065,E2 22555.065} C_VEL
LIN {X 0,Y 479.031,Z 385.93,A -85,B 0,C 180,E1 22554.422,E2 22554.422} C_VEL
LIN {X 0,Y 481.428,Z 344.114,A -85,B 0,C 180,E1 22551.534,E2 22551.534} C_VEL
LIN {X 0,Y 472.656,Z 322.365,A -85,B 0,C 180,E1 22549.135,E2 22549.135} C_VEL
LIN {X 0,Y 465.083,Z 304.995,A -85,B 0,C 180,E1 22546.989,E2 22546.989} C_VEL
LIN {X 0,Y 465.002,Z 304.531,A -85,B 0,C 180,E1 22546.617,E2 22546.617} C_VEL
LIN {X 0,Y 465.014,Z 304.537,A -85,B 0,C 180,E1 22542.969,E2 22542.969} C_VEL
LIN {X 0,Y 464.996,Z 304.563,A -85,B 0,C 180,E1 22539.37,E2 22539.37} C_VEL
LIN {X 0,Y 464.967,Z 304.528,A -85,B 0,C 180,E1 22535.796,E2 22535.796} C_VEL
LIN {X 0,Y 464.973,Z 304.562,A -85,B 0,C 180,E1 22532.082,E2 22532.082} C_VEL
LIN {X 0,Y 465.004,Z 304.561,A -85,B 0,C 180,E1 22528.512,E2 22528.512} C_VEL
LIN {X 0,Y 465.013,Z 304.565,A -85,B 0,C 180,E1 22524.789,E2 22524.789} C_VEL
LIN {X 0,Y 464.971,Z 304.563,A -85,B 0,C 180,E1 22521.31,E2 22521.31} C_VEL
LIN {X 0,Y 464.954,Z 304.56,A -85,B 0,C 180,E1 22517.708,E2 22517.708} C_VEL
LIN {X 0,Y 464.967,Z 304.551,A -85,B 0,C 180,E1 22514.118,E2 22514.118} C_VEL
LIN {X 0,Y 465,Z 304.564,A -85,B 0,C 180,E1 22510.531,E2 22510.531} C_VEL
LIN {X 0,Y 464.972,Z 304.557,A -85,B 0,C 180,E1 22506.916,E2 22506.916} C_VEL
LIN {X 0,Y 464.939,Z 304.558,A -85,B 0,C 180,E1 22503.452,E2 22503.452} C_VEL
LIN {X 0,Y 464.942,Z 304.567,A -85,B 0,C 180,E1 22499.753,E2 22499.753} C_VEL
LIN {X 0,Y 464.97,Z 304.555,A -85,B 0,C 180,E1 22496.177,E2 22496.177} C_VEL
LIN {X 0,Y 464.984,Z 304.556,A -85,B 0,C 180,E1 22492.587,E2 22492.587} C_VEL
LIN {X 0,Y 464.954,Z 304.565,A -85,B 0,C 180,E1 22488.966,E2 22488.966} C_VEL
LIN {X 0,Y 464.943,Z 304.552,A -85,B 0,C 180,E1 22485.397,E2 22485.397} C_VEL
LIN {X 0,Y 464.97,Z 304.559,A -85,B 0,C 180,E1 22481.832,E2 22481.832} C_VEL
LIN {X 0,Y 465.011,Z 304.564,A -85,B 0,C 180,E1 22478.162,E2 22478.162} C_VEL
LIN {X 0,Y 464.988,Z 304.551,A -85,B 0,C 180,E1 22474.528,E2 22474.528} C_VEL
LIN {X 0,Y 464.961,Z 304.56,A -85,B 0,C 180,E1 22471.063,E2 22471.063} C_VEL
LIN {X 0,Y 464.966,Z 304.563,A -85,B 0,C 180,E1 22467.333,E2 22467.333} C_VEL
LIN {X 0,Y 464.996,Z 304.562,A -85,B 0,C 180,E1 22463.738,E2 22463.738} C_VEL
LIN {X 0,Y 465.021,Z 304.562,A -85,B 0,C 180,E1 22460.137,E2 22460.137} C_VEL
LIN {X 0,Y 464.995,Z 304.564,A -85,B 0,C 180,E1 22456.437,E2 22456.437} C_VEL
LIN {X 0,Y 464.975,Z 304.537,A -85,B 0,C 180,E1 22452.804,E2 22452.804} C_VEL
LIN {X 0,Y 464.977,Z 304.538,A -85,B 0,C 180,E1 22449.079,E2 22449.079} C_VEL
LIN {X 0,Y 464.998,Z 304.545,A -85,B 0,C 180,E1 22445.418,E2 22445.418} C_VEL
LIN {X 0,Y 465.022,Z 304.832,A -85,B 0,C 180,E1 22444.843,E2 22444.843} C_VEL
LIN {X 0,Y 471.654,Z 323.172,A -85,B 0,C 180,E1 22442.009,E2 22442.009} C_VEL
LIN {X 0,Y 476.557,Z 338.304,A -85,B 0,C 180,E1 22439.893,E2 22439.893} C_VEL
LIN {X 0,Y 476.607,Z 340.692,A -85,B 0,C 180,E1 22439.699,E2 22439.699} C_VEL
LIN {X 0,Y 480.435,Z 359.218,A -85,B 0,C 180,E1 22439.096,E2 22439.096} C_VEL
LIN {X 0,Y 480.145,Z 380.86,A -85,B 0,C 180,E1 22438.769,E2 22438.769} C_VEL
LIN {X 0,Y 479.198,Z 388.556,A -85,B 0,C 180,E1 22438.717,E2 22438.717} C_VEL
LIN {X 0,Y 473.655,Z 409.052,A -85,B 0,C 180,E1 22438.807,E2 22438.807} C_VEL
LIN {X 0,Y 472.928,Z 415.659,A -85,B 0,C 180,E1 22438.756,E2 22438.756} C_VEL
LIN {X 0,Y 471.37,Z 554.407,A -85,B 0,C 180,E1 22436.659,E2 22436.659} C_VEL
LIN {X 0,Y 470.896,Z 573.572,A -85,B 0,C 180,E1 22436.132,E2 22436.132} C_VEL
LIN {X 0,Y 470.073,Z 591.528,A -85,B 0,C 180,E1 22435.411,E2 22435.411} C_VEL
LIN {X 0,Y 468.963,Z 608.953,A -85,B 0,C 180,E1 22434.475,E2 22434.475} C_VEL
LIN {X 0,Y 467.544,Z 626.01,A -85,B 0,C 180,E1 22433.304,E2 22433.304} C_VEL
LIN {X 0,Y 466.037,Z 641.481,A -85,B 0,C 180,E1 22431.985,E2 22431.985} C_VEL
LIN {X 0,Y 464.431,Z 655.983,A -85,B 0,C 180,E1 22430.477,E2 22430.477} C_VEL
LIN {X 0,Y 462.834,Z 669.456,A -85,B 0,C 180,E1 22428.776,E2 22428.776} C_VEL
LIN {X 0,Y 461.286,Z 681.817,A -85,B 0,C 180,E1 22426.884,E2 22426.884} C_VEL
LIN {X 0,Y 459.958,Z 692.644,A -85,B 0,C 180,E1 22424.863,E2 22424.863} C_VEL
LIN {X 0,Y 458.83,Z 701.997,A -85,B 0,C 180,E1 22422.714,E2 22422.714} C_VEL
LIN {X 0,Y 457.962,Z 709.86,A -85,B 0,C 180,E1 22420.44,E2 22420.44} C_VEL
LIN {X 0,Y 457.353,Z 716.195,A -85,B 0,C 180,E1 22418.043,E2 22418.043} C_VEL
LIN {X 0,Y 456.956,Z 720.742,A -85,B 0,C 180,E1 22415.651,E2 22415.651} C_VEL
LIN {X 0,Y 456.74,Z 723.638,A -85,B 0,C 180,E1 22413.263,E2 22413.263} C_VEL
LIN {X 0,Y 456.661,Z 725.002,A -85,B 0,C 180,E1 22410.753,E2 22410.753} C_VEL
LIN {X 0,Y 456.679,Z 724.697,A -85,B 0,C 180,E1 22408.244,E2 22408.244} C_VEL
LIN {X 0,Y 456.807,Z 722.71,A -85,B 0,C 180,E1 22405.732,E2 22405.732} C_VEL
LIN {X 0,Y 457.102,Z 718.964,A -85,B 0,C 180,E1 22403.217,E2 22403.217} C_VEL
LIN {X 0,Y 457.589,Z 713.653,A -85,B 0,C 180,E1 22400.822,E2 22400.822} C_VEL
LIN {X 0,Y 458.275,Z 706.892,A -85,B 0,C 180,E1 22398.549,E2 22398.549} C_VEL
LIN {X 0,Y 459.214,Z 698.747,A -85,B 0,C 180,E1 22396.4,E2 22396.4} C_VEL
LIN {X 0,Y 460.44,Z 688.616,A -85,B 0,C 180,E1 22394.25,E2 22394.25} C_VEL
LIN {X 0,Y 461.863,Z 677.188,A -85,B 0,C 180,E1 22392.276,E2 22392.276} C_VEL
LIN {X 0,Y 463.439,Z 664.431,A -85,B 0,C 180,E1 22390.464,E2 22390.464} C_VEL
LIN {X 0,Y 465.056,Z 650.47,A -85,B 0,C 180,E1 22388.827,E2 22388.827} C_VEL
LIN {X 0,Y 466.65,Z 635.471,A -85,B 0,C 180,E1 22387.382,E2 22387.382} C_VEL
LIN {X 0,Y 468.035,Z 620.346,A -85,B 0,C 180,E1 22386.187,E2 22386.187} C_VEL
LIN {X 0,Y 469.311,Z 603.926,A -85,B 0,C 180,E1 22385.142,E2 22385.142} C_VEL
LIN {X 0,Y 470.343,Z 586.287,A -85,B 0,C 180,E1 22384.267,E2 22384.267} C_VEL
LIN {X 0,Y 471.079,Z 567.644,A -85,B 0,C 180,E1 22383.591,E2 22383.591} C_VEL
LIN {X 0,Y 471.426,Z 548.714,A -85,B 0,C 180,E1 22383.142,E2 22383.142} C_VEL
LIN {X 0,Y 473.554,Z 359.044,A -85,B 0,C 180,E1 22380.271,E2 22380.271} C_VEL
LIN {X 0,Y 469.391,Z 340.655,A -85,B 0,C 180,E1 22379.622,E2 22379.622} C_VEL
LIN {X 0,Y 463.748,Z 323.819,A -85,B 0,C 180,E1 22377.231,E2 22377.231} C_VEL
LIN {X 0,Y 457.853,Z 308.147,A -85,B 0,C 180,E1 22374.76,E2 22374.76} C_VEL
LIN {X 0,Y 457.088,Z 305.664,A -85,B 0,C 180,E1 22374.304,E2 22374.304} C_VEL
LIN {X 0,Y 457.054,Z 305.524,A -85,B 0,C 180,E1 22370.625,E2 22370.625} C_VEL
LIN {X 0,Y 457.04,Z 305.52,A -85,B 0,C 180,E1 22366.958,E2 22366.958} C_VEL
LIN {X 0,Y 457.046,Z 305.555,A -85,B 0,C 180,E1 22363.215,E2 22363.215} C_VEL
LIN {X 0,Y 457.072,Z 305.554,A -85,B 0,C 180,E1 22359.647,E2 22359.647} C_VEL
LIN {X 0,Y 457.077,Z 305.551,A -85,B 0,C 180,E1 22355.892,E2 22355.892} C_VEL
LIN {X 0,Y 457.052,Z 305.549,A -85,B 0,C 180,E1 22352.262,E2 22352.262} C_VEL
LIN {X 0,Y 457.027,Z 305.548,A -85,B 0,C 180,E1 22348.686,E2 22348.686} C_VEL
LIN {X 0,Y 457.025,Z 305.539,A -85,B 0,C 180,E1 22344.976,E2 22344.976} C_VEL
LIN {X 0,Y 457.054,Z 305.549,A -85,B 0,C 180,E1 22341.428,E2 22341.428} C_VEL
LIN {X 0,Y 457.06,Z 305.546,A -85,B 0,C 180,E1 22337.834,E2 22337.834} C_VEL
LIN {X 0,Y 457.019,Z 305.538,A -85,B 0,C 180,E1 22334.267,E2 22334.267} C_VEL
LIN {X 0,Y 457.007,Z 305.553,A -85,B 0,C 180,E1 22330.59,E2 22330.59} C_VEL
LIN {X 0,Y 457.009,Z 305.555,A -85,B 0,C 180,E1 22326.911,E2 22326.911} C_VEL
LIN {X 0,Y 457.043,Z 305.537,A -85,B 0,C 180,E1 22323.387,E2 22323.387} C_VEL
LIN {X 0,Y 457.031,Z 305.556,A -85,B 0,C 180,E1 22319.75,E2 22319.75} C_VEL
LIN {X 0,Y 457.004,Z 305.546,A -85,B 0,C 180,E1 22316.111,E2 22316.111} C_VEL
LIN {X 0,Y 457.002,Z 305.545,A -85,B 0,C 180,E1 22312.457,E2 22312.457} C_VEL
LIN {X 0,Y 457.026,Z 305.554,A -85,B 0,C 180,E1 22308.9,E2 22308.9} C_VEL
LIN {X 0,Y 457.071,Z 305.542,A -85,B 0,C 180,E1 22305.301,E2 22305.301} C_VEL
LIN {X 0,Y 457.044,Z 305.541,A -85,B 0,C 180,E1 22301.638,E2 22301.638} C_VEL
LIN {X 0,Y 457.024,Z 305.553,A -85,B 0,C 180,E1 22298.031,E2 22298.031} C_VEL
LIN {X 0,Y 457.024,Z 305.554,A -85,B 0,C 180,E1 22294.331,E2 22294.331} C_VEL
LIN {X 0,Y 457.052,Z 305.552,A -85,B 0,C 180,E1 22290.79,E2 22290.79} C_VEL
LIN {X 0,Y 457.075,Z 305.551,A -85,B 0,C 180,E1 22287.138,E2 22287.138} C_VEL
LIN {X 0,Y 457.055,Z 305.511,A -85,B 0,C 180,E1 22283.485,E2 22283.485} C_VEL
LIN {X 0,Y 457.036,Z 305.541,A -85,B 0,C 180,E1 22279.967,E2 22279.967} C_VEL
LIN {X 0,Y 457.042,Z 305.553,A -85,B 0,C 180,E1 22276.212,E2 22276.212} C_VEL
LIN {X 0,Y 457.062,Z 305.676,A -85,B 0,C 180,E1 22273.848,E2 22273.848} C_VEL
LIN {X 0,Y 457.472,Z 307.266,A -85,B 0,C 180,E1 22273.57,E2 22273.57} C_VEL
LIN {X 0,Y 462.54,Z 318.305,A -85,B 0,C 180,E1 22272.145,E2 22272.145} C_VEL
LIN {X 0,Y 470.549,Z 337.177,A -85,B 0,C 180,E1 22269.908,E2 22269.908} C_VEL
LIN {X 0,Y 474.52,Z 347.604,A -85,B 0,C 180,E1 22268.774,E2 22268.774} C_VEL
LIN {X 0,Y 472.12,Z 386.495,A -85,B 0,C 180,E1 22266.081,E2 22266.081} C_VEL
LIN {X 0,Y 475.165,Z 413.726,A -85,B 0,C 180,E1 22265.344,E2 22265.344} C_VEL
LIN {X 0,Y 470.643,Z 641.643,A -85,B 0,C 180,E1 22261.463,E2 22261.463} C_VEL
LIN {X 0,Y 469.666,Z 663.065,A -85,B 0,C 180,E1 22260.926,E2 22260.926} C_VEL
LIN {X 0,Y 468.44,Z 683.801,A -85,B 0,C 180,E1 22260.18,E2 22260.18} C_VEL
LIN {X 0,Y 467.029,Z 704.15,A -85,B 0,C 180,E1 22259.216,E2 22259.216} C_VEL
LIN {X 0,Y 465.511,Z 724.195,A -85,B 0,C 180,E1 22258.021,E2 22258.021} C_VEL
LIN {X 0,Y 463.96,Z 743.389,A -85,B 0,C 180,E1 22256.631,E2 22256.631} C_VEL
LIN {X 0,Y 462.458,Z 761.5,A -85,B 0,C 180,E1 22255.056,E2 22255.056} C_VEL
LIN {X 0,Y 460.987,Z 778.905,A -85,B 0,C 180,E1 22253.25,E2 22253.25} C_VEL
LIN {X 0,Y 459.681,Z 794.746,A -85,B 0,C 180,E1 22251.299,E2 22251.299} C_VEL
LIN {X 0,Y 458.601,Z 808.779,A -85,B 0,C 180,E1 22249.259,E2 22249.259} C_VEL
LIN {X 0,Y 457.674,Z 821.782,A -85,B 0,C 180,E1 22247.022,E2 22247.022} C_VEL
LIN {X 0,Y 456.995,Z 832.984,A -85,B 0,C 180,E1 22244.702,E2 22244.702} C_VEL
LIN {X 0,Y 456.51,Z 842.323,A -85,B 0,C 180,E1 22242.356,E2 22242.356} C_VEL
LIN {X 0,Y 456.225,Z 849.97,A -85,B 0,C 180,E1 22239.97,E2 22239.97} C_VEL
LIN {X 0,Y 456.07,Z 855.847,A -85,B 0,C 180,E1 22237.558,E2 22237.558} C_VEL
LIN {X 0,Y 456.011,Z 860.066,A -85,B 0,C 180,E1 22235.158,E2 22235.158} C_VEL
LIN {X 0,Y 455.994,Z 862.711,A -85,B 0,C 180,E1 22232.765,E2 22232.765} C_VEL
LIN {X 0,Y 455.985,Z 863.702,A -85,B 0,C 180,E1 22230.377,E2 22230.377} C_VEL
LIN {X 0,Y 455.989,Z 863.084,A -85,B 0,C 180,E1 22227.864,E2 22227.864} C_VEL
LIN {X 0,Y 455.993,Z 860.931,A -85,B 0,C 180,E1 22225.473,E2 22225.473} C_VEL
LIN {X 0,Y 456.052,Z 857.151,A -85,B 0,C 180,E1 22223.074,E2 22223.074} C_VEL
LIN {X 0,Y 456.182,Z 851.659,A -85,B 0,C 180,E1 22220.666,E2 22220.666} C_VEL
LIN {X 0,Y 456.429,Z 844.406,A -85,B 0,C 180,E1 22218.245,E2 22218.245} C_VEL
LIN {X 0,Y 456.835,Z 835.774,A -85,B 0,C 180,E1 22215.94,E2 22215.94} C_VEL
LIN {X 0,Y 457.454,Z 825.167,A -85,B 0,C 180,E1 22213.623,E2 22213.623} C_VEL
LIN {X 0,Y 458.281,Z 813.035,A -85,B 0,C 180,E1 22211.426,E2 22211.426} C_VEL
LIN {X 0,Y 459.3,Z 799.458,A -85,B 0,C 180,E1 22209.35,E2 22209.35} C_VEL
LIN {X 0,Y 460.592,Z 783.658,A -85,B 0,C 180,E1 22207.308,E2 22207.308} C_VEL
LIN {X 0,Y 462.014,Z 766.602,A -85,B 0,C 180,E1 22205.449,E2 22205.449} C_VEL
LIN {X 0,Y 463.508,Z 748.798,A -85,B 0,C 180,E1 22203.815,E2 22203.815} C_VEL
LIN {X 0,Y 465.015,Z 730.37,A -85,B 0,C 180,E1 22202.397,E2 22202.397} C_VEL
LIN {X 0,Y 466.529,Z 711.204,A -85,B 0,C 180,E1 22201.171,E2 22201.171} C_VEL
LIN {X 0,Y 468.035,Z 689.959,A -85,B 0,C 180,E1 22200.079,E2 22200.079} C_VEL
LIN {X 0,Y 469.413,Z 668.411,A -85,B 0,C 180,E1 22199.239,E2 22199.239} C_VEL
LIN {X 0,Y 470.478,Z 646.724,A -85,B 0,C 180,E1 22198.641,E2 22198.641} C_VEL
LIN {X 0,Y 471.694,Z 588.524,A -85,B 0,C 180,E1 22197.624,E2 22197.624} C_VEL
LIN {X 0,Y 475.091,Z 411.358,A -85,B 0,C 180,E1 22194.607,E2 22194.607} C_VEL
LIN {X 0,Y 472.05,Z 385.383,A -85,B 0,C 180,E1 22193.875,E2 22193.875} C_VEL
LIN {X 0,Y 474.446,Z 347.142,A -85,B 0,C 180,E1 22191.189,E2 22191.189} C_VEL
LIN {X 0,Y 466.077,Z 326.392,A -85,B 0,C 180,E1 22188.85,E2 22188.85} C_VEL
LIN {X 0,Y 458.118,Z 308.607,A -85,B 0,C 180,E1 22186.617,E2 22186.617} C_VEL
LIN {X 0,Y 457.083,Z 305.806,A -85,B 0,C 180,E1 22186.209,E2 22186.209} C_VEL
LIN {X 0,Y 457.043,Z 305.557,A -85,B 0,C 180,E1 22184.149,E2 22184.149} C_VEL
LIN {X 0,Y 457.06,Z 305.526,A -85,B 0,C 180,E1 22180.52,E2 22180.52} C_VEL
LIN {X 0,Y 457.073,Z 305.515,A -85,B 0,C 180,E1 22176.982,E2 22176.982} C_VEL
LIN {X 0,Y 457.051,Z 305.55,A -85,B 0,C 180,E1 22173.305,E2 22173.305} C_VEL
LIN {X 0,Y 457.029,Z 305.555,A -85,B 0,C 180,E1 22169.715,E2 22169.715} C_VEL
LIN {X 0,Y 457.033,Z 305.555,A -85,B 0,C 180,E1 22166.086,E2 22166.086} C_VEL
LIN {X 0,Y 457.062,Z 305.542,A -85,B 0,C 180,E1 22162.509,E2 22162.509} C_VEL
LIN {X 0,Y 457.058,Z 305.541,A -85,B 0,C 180,E1 22158.89,E2 22158.89} C_VEL
LIN {X 0,Y 457.025,Z 305.554,A -85,B 0,C 180,E1 22155.254,E2 22155.254} C_VEL
LIN {X 0,Y 457.01,Z 305.554,A -85,B 0,C 180,E1 22151.612,E2 22151.612} C_VEL
LIN {X 0,Y 457.014,Z 305.542,A -85,B 0,C 180,E1 22147.922,E2 22147.922} C_VEL
LIN {X 0,Y 457.048,Z 305.547,A -85,B 0,C 180,E1 22144.391,E2 22144.391} C_VEL
LIN {X 0,Y 457.051,Z 305.55,A -85,B 0,C 180,E1 22140.626,E2 22140.626} C_VEL
LIN {X 0,Y 457.007,Z 305.539,A -85,B 0,C 180,E1 22136.99,E2 22136.99} C_VEL
LIN {X 0,Y 456.998,Z 305.555,A -85,B 0,C 180,E1 22133.349,E2 22133.349} C_VEL
LIN {X 0,Y 457.008,Z 305.554,A -85,B 0,C 180,E1 22129.665,E2 22129.665} C_VEL
LIN {X 0,Y 457.042,Z 305.536,A -85,B 0,C 180,E1 22126.075,E2 22126.075} C_VEL
LIN {X 0,Y 457.057,Z 305.552,A -85,B 0,C 180,E1 22122.429,E2 22122.429} C_VEL
LIN {X 0,Y 457.025,Z 305.548,A -85,B 0,C 180,E1 22118.839,E2 22118.839} C_VEL
LIN {X 0,Y 457.016,Z 305.539,A -85,B 0,C 180,E1 22115.218,E2 22115.218} C_VEL
LIN {X 0,Y 457.032,Z 305.548,A -85,B 0,C 180,E1 22111.575,E2 22111.575} C_VEL
LIN {X 0,Y 457.074,Z 305.551,A -85,B 0,C 180,E1 22108.036,E2 22108.036} C_VEL
LIN {X 0,Y 457.057,Z 305.553,A -85,B 0,C 180,E1 22104.415,E2 22104.415} C_VEL
LIN {X 0,Y 457.035,Z 305.553,A -85,B 0,C 180,E1 22100.784,E2 22100.784} C_VEL
LIN {X 0,Y 457.036,Z 305.554,A -85,B 0,C 180,E1 22097.127,E2 22097.127} C_VEL
LIN {X 0,Y 457.055,Z 305.514,A -85,B 0,C 180,E1 22093.557,E2 22093.557} C_VEL
LIN {X 0,Y 457.079,Z 305.533,A -85,B 0,C 180,E1 22089.86,E2 22089.86} C_VEL
LIN {X 0,Y 457.07,Z 305.551,A -85,B 0,C 180,E1 22086.176,E2 22086.176} C_VEL
LIN {X 0,Y 457.103,Z 305.805,A -85,B 0,C 180,E1 22085.54,E2 22085.54} C_VEL
LIN {X 0,Y 463.769,Z 323.915,A -85,B 0,C 180,E1 22082.659,E2 22082.659} C_VEL
LIN {X 0,Y 469.458,Z 340.836,A -85,B 0,C 180,E1 22080.272,E2 22080.272} C_VEL
LIN {X 0,Y 473.675,Z 360.592,A -85,B 0,C 180,E1 22079.595,E2 22079.595} C_VEL
LIN {X 0,Y 472.928,Z 415.659,A -85,B 0,C 180,E1 22078.756,E2 22078.756} C_VEL
LIN {X 0,Y 471.972,Z 423.356,A -85,B 0,C 180,E1 22078.706,E2 22078.706} C_VEL
LIN {X 0,Y 466.393,Z 443.845,A -85,B 0,C 180,E1 22078.803,E2 22078.803} C_VEL
LIN {X 0,Y 465.674,Z 450.451,A -85,B 0,C 180,E1 22078.752,E2 22078.752} C_VEL
LIN {X 0,Y 464.448,Z 555.437,A -85,B 0,C 180,E1 22077.136,E2 22077.136} C_VEL
LIN {X 0,Y 463.939,Z 574.591,A -85,B 0,C 180,E1 22076.601,E2 22076.601} C_VEL
LIN {X 0,Y 463.055,Z 592.759,A -85,B 0,C 180,E1 22075.859,E2 22075.859} C_VEL
LIN {X 0,Y 461.864,Z 610.346,A -85,B 0,C 180,E1 22074.896,E2 22074.896} C_VEL
LIN {X 0,Y 460.428,Z 626.775,A -85,B 0,C 180,E1 22073.754,E2 22073.754} C_VEL
LIN {X 0,Y 458.829,Z 642.304,A -85,B 0,C 180,E1 22072.417,E2 22072.417} C_VEL
LIN {X 0,Y 457.058,Z 657.387,A -85,B 0,C 180,E1 22070.823,E2 22070.823} C_VEL
LIN {X 0,Y 455.37,Z 670.816,A -85,B 0,C 180,E1 22069.096,E2 22069.096} C_VEL
LIN {X 0,Y 453.728,Z 683.14,A -85,B 0,C 180,E1 22067.174,E2 22067.174} C_VEL
LIN {X 0,Y 452.311,Z 693.94,A -85,B 0,C 180,E1 22065.12,E2 22065.12} C_VEL
LIN {X 0,Y 451.104,Z 703.269,A -85,B 0,C 180,E1 22062.936,E2 22062.936} C_VEL
LIN {X 0,Y 450.168,Z 711.111,A -85,B 0,C 180,E1 22060.623,E2 22060.623} C_VEL
LIN {X 0,Y 449.509,Z 717.445,A -85,B 0,C 180,E1 22058.176,E2 22058.176} C_VEL
LIN {X 0,Y 449.079,Z 721.959,A -85,B 0,C 180,E1 22055.75,E2 22055.75} C_VEL
LIN {X 0,Y 448.842,Z 724.845,A -85,B 0,C 180,E1 22053.32,E2 22053.32} C_VEL
LIN {X 0,Y 448.752,Z 726.203,A -85,B 0,C 180,E1 22050.766,E2 22050.766} C_VEL
LIN {X 0,Y 448.772,Z 725.9,A -85,B 0,C 180,E1 22048.213,E2 22048.213} C_VEL
LIN {X 0,Y 448.915,Z 723.921,A -85,B 0,C 180,E1 22045.657,E2 22045.657} C_VEL
LIN {X 0,Y 449.237,Z 720.186,A -85,B 0,C 180,E1 22043.097,E2 22043.097} C_VEL
LIN {X 0,Y 449.766,Z 714.892,A -85,B 0,C 180,E1 22040.661,E2 22040.661} C_VEL
LIN {X 0,Y 450.51,Z 708.15,A -85,B 0,C 180,E1 22038.348,E2 22038.348} C_VEL
LIN {X 0,Y 451.518,Z 700.026,A -85,B 0,C 180,E1 22036.164,E2 22036.164} C_VEL
LIN {X 0,Y 452.828,Z 689.922,A -85,B 0,C 180,E1 22033.979,E2 22033.979} C_VEL
LIN {X 0,Y 454.274,Z 679.021,A -85,B 0,C 180,E1 22032.053,E2 22032.053} C_VEL
LIN {X 0,Y 455.974,Z 666.102,A -85,B 0,C 180,E1 22030.172,E2 22030.172} C_VEL
LIN {X 0,Y 457.635,Z 652.624,A -85,B 0,C 180,E1 22028.552,E2 22028.552} C_VEL
LIN {X 0,Y 459.324,Z 637.67,A -85,B 0,C 180,E1 22027.068,E2 22027.068} C_VEL
LIN {X 0,Y 460.868,Z 621.935,A -85,B 0,C 180,E1 22025.794,E2 22025.794} C_VEL
LIN {X 0,Y 462.244,Z 605.266,A -85,B 0,C 180,E1 22024.711,E2 22024.711} C_VEL
LIN {X 0,Y 463.346,Z 587.531,A -85,B 0,C 180,E1 22023.815,E2 22023.815} C_VEL
LIN {X 0,Y 464.133,Z 568.86,A -85,B 0,C 180,E1 22023.125,E2 22023.125} C_VEL
LIN {X 0,Y 464.508,Z 549.822,A -85,B 0,C 180,E1 22022.664,E2 22022.664} C_VEL
LIN {X 0,Y 466.839,Z 360.55,A -85,B 0,C 180,E1 22019.758,E2 22019.758} C_VEL
LIN {X 0,Y 463.216,Z 344.477,A -85,B 0,C 180,E1 22019.185,E2 22019.185} C_VEL
LIN {X 0,Y 461.228,Z 340.497,A -85,B 0,C 180,E1 22018.903,E2 22018.903} C_VEL
LIN {X 0,Y 454.943,Z 322.197,A -85,B 0,C 180,E1 22016.177,E2 22016.177} C_VEL
LIN {X 0,Y 449.159,Z 306.761,A -85,B 0,C 180,E1 22013.614,E2 22013.614} C_VEL
LIN {X 0,Y 449.139,Z 306.517,A -85,B 0,C 180,E1 22010.125,E2 22010.125} C_VEL
LIN {X 0,Y 449.113,Z 306.501,A -85,B 0,C 180,E1 22006.534,E2 22006.534} C_VEL
LIN {X 0,Y 449.102,Z 306.543,A -85,B 0,C 180,E1 22002.908,E2 22002.908} C_VEL
LIN {X 0,Y 449.105,Z 306.541,A -85,B 0,C 180,E1 21999.218,E2 21999.218} C_VEL
LIN {X 0,Y 449.122,Z 306.541,A -85,B 0,C 180,E1 21995.525,E2 21995.525} C_VEL
LIN {X 0,Y 449.14,Z 306.54,A -85,B 0,C 180,E1 21991.748,E2 21991.748} C_VEL
LIN {X 0,Y 449.128,Z 306.534,A -85,B 0,C 180,E1 21988.017,E2 21988.017} C_VEL
LIN {X 0,Y 449.095,Z 306.526,A -85,B 0,C 180,E1 21984.323,E2 21984.323} C_VEL
LIN {X 0,Y 449.08,Z 306.536,A -85,B 0,C 180,E1 21980.733,E2 21980.733} C_VEL
LIN {X 0,Y 449.088,Z 306.544,A -85,B 0,C 180,E1 21977.091,E2 21977.091} C_VEL
LIN {X 0,Y 449.12,Z 306.525,A -85,B 0,C 180,E1 21973.519,E2 21973.519} C_VEL
LIN {X 0,Y 449.112,Z 306.53,A -85,B 0,C 180,E1 21969.742,E2 21969.742} C_VEL
LIN {X 0,Y 449.07,Z 306.544,A -85,B 0,C 180,E1 21966.264,E2 21966.264} C_VEL
LIN {X 0,Y 449.057,Z 306.529,A -85,B 0,C 180,E1 21962.553,E2 21962.553} C_VEL
LIN {X 0,Y 449.072,Z 306.539,A -85,B 0,C 180,E1 21958.98,E2 21958.98} C_VEL
LIN {X 0,Y 449.104,Z 306.54,A -85,B 0,C 180,E1 21955.275,E2 21955.275} C_VEL
LIN {X 0,Y 449.099,Z 306.526,A -85,B 0,C 180,E1 21951.68,E2 21951.68} C_VEL
LIN {X 0,Y 449.077,Z 306.544,A -85,B 0,C 180,E1 21948.05,E2 21948.05} C_VEL
LIN {X 0,Y 449.074,Z 306.544,A -85,B 0,C 180,E1 21944.371,E2 21944.371} C_VEL
LIN {X 0,Y 449.09,Z 306.536,A -85,B 0,C 180,E1 21940.729,E2 21940.729} C_VEL
LIN {X 0,Y 449.126,Z 306.527,A -85,B 0,C 180,E1 21937.071,E2 21937.071} C_VEL
LIN {X 0,Y 449.124,Z 306.531,A -85,B 0,C 180,E1 21933.419,E2 21933.419} C_VEL
LIN {X 0,Y 449.094,Z 306.541,A -85,B 0,C 180,E1 21929.938,E2 21929.938} C_VEL
LIN {X 0,Y 449.093,Z 306.536,A -85,B 0,C 180,E1 21926.179,E2 21926.179} C_VEL
LIN {X 0,Y 449.098,Z 306.518,A -85,B 0,C 180,E1 21922.409,E2 21922.409} C_VEL
LIN {X 0,Y 449.129,Z 306.502,A -85,B 0,C 180,E1 21918.802,E2 21918.802} C_VEL
LIN {X 0,Y 449.137,Z 306.52,A -85,B 0,C 180,E1 21915.065,E2 21915.065} C_VEL
LIN {X 0,Y 449.164,Z 306.836,A -85,B 0,C 180,E1 21914.547,E2 21914.547} C_VEL
LIN {X 0,Y 450.611,Z 310.296,A -85,B 0,C 180,E1 21914.035,E2 21914.035} C_VEL
LIN {X 0,Y 459.097,Z 329.386,A -85,B 0,C 180,E1 21911.574,E2 21911.574} C_VEL
LIN {X 0,Y 467.271,Z 349.616,A -85,B 0,C 180,E1 21909.231,E2 21909.231} C_VEL
LIN {X 0,Y 467.455,Z 351.849,A -85,B 0,C 180,E1 21909.043,E2 21909.043} C_VEL
LIN {X 0,Y 465.163,Z 385.883,A -85,B 0,C 180,E1 21906.644,E2 21906.644} C_VEL
LIN {X 0,Y 468.361,Z 414.894,A -85,B 0,C 180,E1 21905.843,E2 21905.843} C_VEL
LIN {X 0,Y 463.596,Z 639.784,A -85,B 0,C 180,E1 21901.953,E2 21901.953} C_VEL
LIN {X 0,Y 462.57,Z 661.56,A -85,B 0,C 180,E1 21901.407,E2 21901.407} C_VEL
LIN {X 0,Y 461.202,Z 682.982,A -85,B 0,C 180,E1 21900.627,E2 21900.627} C_VEL
LIN {X 0,Y 459.699,Z 703.09,A -85,B 0,C 180,E1 21899.657,E2 21899.657} C_VEL
LIN {X 0,Y 458.115,Z 722.498,A -85,B 0,C 180,E1 21898.481,E2 21898.481} C_VEL
LIN {X 0,Y 456.462,Z 741.224,A -85,B 0,C 180,E1 21897.104,E2 21897.104} C_VEL
LIN {X 0,Y 454.747,Z 760.543,A -85,B 0,C 180,E1 21895.387,E2 21895.387} C_VEL
LIN {X 0,Y 453.188,Z 778.072,A -85,B 0,C 180,E1 21893.536,E2 21893.536} C_VEL
LIN {X 0,Y 451.78,Z 794.389,A -85,B 0,C 180,E1 21891.485,E2 21891.485} C_VEL
LIN {X 0,Y 450.61,Z 808.971,A -85,B 0,C 180,E1 21889.306,E2 21889.306} C_VEL
LIN {X 0,Y 449.729,Z 820.861,A -85,B 0,C 180,E1 21887.198,E2 21887.198} C_VEL
LIN {X 0,Y 449.033,Z 832.082,A -85,B 0,C 180,E1 21884.837,E2 21884.837} C_VEL
LIN {X 0,Y 448.55,Z 841.271,A -85,B 0,C 180,E1 21882.487,E2 21882.487} C_VEL
LIN {X 0,Y 448.267,Z 849.018,A -85,B 0,C 180,E1 21880.019,E2 21880.019} C_VEL
LIN {X 0,Y 448.128,Z 854.858,A -85,B 0,C 180,E1 21877.564,E2 21877.564} C_VEL
LIN {X 0,Y 448.085,Z 859.007,A -85,B 0,C 180,E1 21875.121,E2 21875.121} C_VEL
LIN {X 0,Y 448.079,Z 861.577,A -85,B 0,C 180,E1 21872.686,E2 21872.686} C_VEL
LIN {X 0,Y 448.08,Z 862.524,A -85,B 0,C 180,E1 21870.256,E2 21870.256} C_VEL
LIN {X 0,Y 448.076,Z 861.878,A -85,B 0,C 180,E1 21867.826,E2 21867.826} C_VEL
LIN {X 0,Y 448.072,Z 859.704,A -85,B 0,C 180,E1 21865.392,E2 21865.392} C_VEL
LIN {X 0,Y 448.118,Z 855.896,A -85,B 0,C 180,E1 21862.951,E2 21862.951} C_VEL
LIN {X 0,Y 448.246,Z 850.357,A -85,B 0,C 180,E1 21860.499,E2 21860.499} C_VEL
LIN {X 0,Y 448.482,Z 843.042,A -85,B 0,C 180,E1 21858.034,E2 21858.034} C_VEL
LIN {X 0,Y 448.908,Z 834.248,A -85,B 0,C 180,E1 21855.668,E2 21855.668} C_VEL
LIN {X 0,Y 449.544,Z 823.619,A -85,B 0,C 180,E1 21853.327,E2 21853.327} C_VEL
LIN {X 0,Y 450.454,Z 810.898,A -85,B 0,C 180,E1 21851.01,E2 21851.01} C_VEL
LIN {X 0,Y 451.572,Z 796.731,A -85,B 0,C 180,E1 21848.845,E2 21848.845} C_VEL
LIN {X 0,Y 452.889,Z 781.387,A -85,B 0,C 180,E1 21846.861,E2 21846.861} C_VEL
LIN {X 0,Y 454.387,Z 764.479,A -85,B 0,C 180,E1 21845.009,E2 21845.009} C_VEL
LIN {X 0,Y 456.049,Z 745.912,A -85,B 0,C 180,E1 21843.292,E2 21843.292} C_VEL
LIN {X 0,Y 457.692,Z 727.212,A -85,B 0,C 180,E1 21841.845,E2 21841.845} C_VEL
LIN {X 0,Y 459.337,Z 707.762,A -85,B 0,C 180,E1 21840.604,E2 21840.604} C_VEL
LIN {X 0,Y 460.87,Z 687.741,A -85,B 0,C 180,E1 21839.576,E2 21839.576} C_VEL
LIN {X 0,Y 462.289,Z 666.752,A -85,B 0,C 180,E1 21838.753,E2 21838.753} C_VEL
LIN {X 0,Y 463.451,Z 644.624,A -85,B 0,C 180,E1 21838.143,E2 21838.143} C_VEL
LIN {X 0,Y 468.168,Z 423.727,A -85,B 0,C 180,E1 21834.308,E2 21834.308} C_VEL
LIN {X 0,Y 468.187,Z 411.753,A -85,B 0,C 180,E1 21834.086,E2 21834.086} C_VEL
LIN {X 0,Y 465.121,Z 384.724,A -85,B 0,C 180,E1 21833.302,E2 21833.302} C_VEL
LIN {X 0,Y 467.47,Z 350.191,A -85,B 0,C 180,E1 21830.836,E2 21830.836} C_VEL
LIN {X 0,Y 459.285,Z 329.892,A -85,B 0,C 180,E1 21828.493,E2 21828.493} C_VEL
LIN {X 0,Y 451.764,Z 313.011,A -85,B 0,C 180,E1 21826.33,E2 21826.33} C_VEL
LIN {X 0,Y 449.172,Z 306.891,A -85,B 0,C 180,E1 21825.479,E2 21825.479} C_VEL
LIN {X 0,Y 449.136,Z 306.521,A -85,B 0,C 180,E1 21824.886,E2 21824.886} C_VEL
LIN {X 0,Y 449.13,Z 306.502,A -85,B 0,C 180,E1 21821.198,E2 21821.198} C_VEL
LIN {X 0,Y 449.1,Z 306.518,A -85,B 0,C 180,E1 21817.574,E2 21817.574} C_VEL
LIN {X 0,Y 449.093,Z 306.537,A -85,B 0,C 180,E1 21813.821,E2 21813.821} C_VEL
LIN {X 0,Y 449.096,Z 306.542,A -85,B 0,C 180,E1 21810.062,E2 21810.062} C_VEL
LIN {X 0,Y 449.121,Z 306.533,A -85,B 0,C 180,E1 21806.501,E2 21806.501} C_VEL
LIN {X 0,Y 449.138,Z 306.526,A -85,B 0,C 180,E1 21802.79,E2 21802.79} C_VEL
LIN {X 0,Y 449.102,Z 306.533,A -85,B 0,C 180,E1 21799.103,E2 21799.103} C_VEL
LIN {X 0,Y 449.077,Z 306.543,A -85,B 0,C 180,E1 21795.496,E2 21795.496} C_VEL
LIN {X 0,Y 449.072,Z 306.543,A -85,B 0,C 180,E1 21791.689,E2 21791.689} C_VEL
LIN {X 0,Y 449.083,Z 306.529,A -85,B 0,C 180,E1 21788.063,E2 21788.063} C_VEL
LIN {X 0,Y 449.113,Z 306.537,A -85,B 0,C 180,E1 21784.469,E2 21784.469} C_VEL
LIN {X 0,Y 449.111,Z 306.539,A -85,B 0,C 180,E1 21780.638,E2 21780.638} C_VEL
LIN {X 0,Y 449.073,Z 306.527,A -85,B 0,C 180,E1 21776.937,E2 21776.937} C_VEL
LIN {X 0,Y 449.06,Z 306.544,A -85,B 0,C 180,E1 21773.351,E2 21773.351} C_VEL
LIN {X 0,Y 449.067,Z 306.543,A -85,B 0,C 180,E1 21769.61,E2 21769.61} C_VEL
LIN {X 0,Y 449.091,Z 306.525,A -85,B 0,C 180,E1 21765.955,E2 21765.955} C_VEL
LIN {X 0,Y 449.124,Z 306.538,A -85,B 0,C 180,E1 21762.327,E2 21762.327} C_VEL
LIN {X 0,Y 449.106,Z 306.537,A -85,B 0,C 180,E1 21758.585,E2 21758.585} C_VEL
LIN {X 0,Y 449.081,Z 306.527,A -85,B 0,C 180,E1 21754.974,E2 21754.974} C_VEL
LIN {X 0,Y 449.083,Z 306.537,A -85,B 0,C 180,E1 21751.255,E2 21751.255} C_VEL
LIN {X 0,Y 449.108,Z 306.54,A -85,B 0,C 180,E1 21747.702,E2 21747.702} C_VEL
LIN {X 0,Y 449.135,Z 306.541,A -85,B 0,C 180,E1 21744.005,E2 21744.005} C_VEL
LIN {X 0,Y 449.131,Z 306.544,A -85,B 0,C 180,E1 21740.288,E2 21740.288} C_VEL
LIN {X 0,Y 449.102,Z 306.545,A -85,B 0,C 180,E1 21736.708,E2 21736.708} C_VEL
LIN {X 0,Y 449.097,Z 306.508,A -85,B 0,C 180,E1 21732.942,E2 21732.942} C_VEL
LIN {X 0,Y 449.106,Z 306.512,A -85,B 0,C 180,E1 21729.216,E2 21729.216} C_VEL
LIN {X 0,Y 449.165,Z 306.808,A -85,B 0,C 180,E1 21726.266,E2 21726.266} C_VEL
LIN {X 0,Y 455.602,Z 324.164,A -85,B 0,C 180,E1 21723.424,E2 21723.424} C_VEL
LIN {X 0,Y 461.389,Z 340.979,A -85,B 0,C 180,E1 21720.949,E2 21720.949} C_VEL
LIN {X 0,Y 463.678,Z 345.93,A -85,B 0,C 180,E1 21720.654,E2 21720.654} C_VEL
LIN {X 0,Y 466.947,Z 362.206,A -85,B 0,C 180,E1 21720.105,E2 21720.105} C_VEL
LIN {X 0,Y 465.674,Z 450.451,A -85,B 0,C 180,E1 21718.752,E2 21718.752} C_VEL
LIN {X 0,Y 464.731,Z 458.149,A -85,B 0,C 180,E1 21718.701,E2 21718.701} C_VEL
LIN {X 0,Y 459.143,Z 478.637,A -85,B 0,C 180,E1 21718.803,E2 21718.803} C_VEL
LIN {X 0,Y 458.427,Z 485.244,A -85,B 0,C 180,E1 21718.751,E2 21718.751} C_VEL
LIN {X 0,Y 457.554,Z 556.603,A -85,B 0,C 180,E1 21717.624,E2 21717.624} C_VEL
LIN {X 0,Y 457.008,Z 575.637,A -85,B 0,C 180,E1 21717.082,E2 21717.082} C_VEL
LIN {X 0,Y 456.071,Z 593.857,A -85,B 0,C 180,E1 21716.326,E2 21716.326} C_VEL
LIN {X 0,Y 454.859,Z 610.95,A -85,B 0,C 180,E1 21715.381,E2 21715.381} C_VEL
LIN {X 0,Y 453.336,Z 627.514,A -85,B 0,C 180,E1 21714.219,E2 21714.219} C_VEL
LIN {X 0,Y 451.566,Z 643.756,A -85,B 0,C 180,E1 21712.797,E2 21712.797} C_VEL
LIN {X 0,Y 449.774,Z 658.25,A -85,B 0,C 180,E1 21711.244,E2 21711.244} C_VEL
LIN {X 0,Y 447.917,Z 672.162,A -85,B 0,C 180,E1 21709.426,E2 21709.426} C_VEL
LIN {X 0,Y 446.18,Z 684.452,A -85,B 0,C 180,E1 21707.474,E2 21707.474} C_VEL
LIN {X 0,Y 444.671,Z 695.225,A -85,B 0,C 180,E1 21705.386,E2 21705.386} C_VEL
LIN {X 0,Y 443.385,Z 704.531,A -85,B 0,C 180,E1 21703.165,E2 21703.165} C_VEL
LIN {X 0,Y 442.379,Z 712.355,A -85,B 0,C 180,E1 21700.812,E2 21700.812} C_VEL
LIN {X 0,Y 441.688,Z 718.493,A -85,B 0,C 180,E1 21698.408,E2 21698.408} C_VEL
LIN {X 0,Y 441.222,Z 722.989,A -85,B 0,C 180,E1 21695.983,E2 21695.983} C_VEL
LIN {X 0,Y 440.953,Z 725.95,A -85,B 0,C 180,E1 21693.51,E2 21693.51} C_VEL
LIN {X 0,Y 440.844,Z 727.386,A -85,B 0,C 180,E1 21690.91,E2 21690.91} C_VEL
LIN {X 0,Y 440.863,Z 727.163,A -85,B 0,C 180,E1 21688.311,E2 21688.311} C_VEL
LIN {X 0,Y 441.011,Z 725.273,A -85,B 0,C 180,E1 21685.709,E2 21685.709} C_VEL
LIN {X 0,Y 441.351,Z 721.635,A -85,B 0,C 180,E1 21683.104,E2 21683.104} C_VEL
LIN {X 0,Y 441.945,Z 716.126,A -85,B 0,C 180,E1 21680.494,E2 21680.494} C_VEL
LIN {X 0,Y 442.749,Z 709.4,A -85,B 0,C 180,E1 21678.141,E2 21678.141} C_VEL
LIN {X 0,Y 443.829,Z 701.296,A -85,B 0,C 180,E1 21675.919,E2 21675.919} C_VEL
LIN {X 0,Y 445.225,Z 691.214,A -85,B 0,C 180,E1 21673.697,E2 21673.697} C_VEL
LIN {X 0,Y 446.762,Z 680.343,A -85,B 0,C 180,E1 21671.741,E2 21671.741} C_VEL
LIN {X 0,Y 448.47,Z 668.121,A -85,B 0,C 180,E1 21669.92,E2 21669.92} C_VEL
LIN {X 0,Y 450.259,Z 654.459,A -85,B 0,C 180,E1 21668.233,E2 21668.233} C_VEL
LIN {X 0,Y 452.093,Z 639.146,A -85,B 0,C 180,E1 21666.68,E2 21666.68} C_VEL
LIN {X 0,Y 453.805,Z 622.633,A -85,B 0,C 180,E1 21665.323,E2 21665.323} C_VEL
LIN {X 0,Y 455.262,Z 605.77,A -85,B 0,C 180,E1 21664.218,E2 21664.218} C_VEL
LIN {X 0,Y 456.418,Z 588.013,A -85,B 0,C 180,E1 21663.316,E2 21663.316} C_VEL
LIN {X 0,Y 457.233,Z 569.486,A -85,B 0,C 180,E1 21662.627,E2 21662.627} C_VEL
LIN {X 0,Y 457.625,Z 550.546,A -85,B 0,C 180,E1 21662.164,E2 21662.164} C_VEL
LIN {X 0,Y 460.162,Z 362.043,A -85,B 0,C 180,E1 21659.23,E2 21659.23} C_VEL
LIN {X 0,Y 457.006,Z 348.141,A -85,B 0,C 180,E1 21658.719,E2 21658.719} C_VEL
LIN {X 0,Y 453.359,Z 341.115,A -85,B 0,C 180,E1 21658.234,E2 21658.234} C_VEL
LIN {X 0,Y 447.108,Z 323.226,A -85,B 0,C 180,E1 21655.495,E2 21655.495} C_VEL
LIN {X 0,Y 442.158,Z 310.486,A -85,B 0,C 180,E1 21653.347,E2 21653.347} C_VEL
LIN {X 0,Y 441.194,Z 307.667,A -85,B 0,C 180,E1 21652.811,E2 21652.811} C_VEL
LIN {X 0,Y 441.17,Z 307.534,A -85,B 0,C 180,E1 21649.083,E2 21649.083} C_VEL
LIN {X 0,Y 441.171,Z 307.493,A -85,B 0,C 180,E1 21645.368,E2 21645.368} C_VEL
LIN {X 0,Y 441.191,Z 307.519,A -85,B 0,C 180,E1 21641.596,E2 21641.596} C_VEL
LIN {X 0,Y 441.202,Z 307.516,A -85,B 0,C 180,E1 21637.89,E2 21637.89} C_VEL
LIN {X 0,Y 441.181,Z 307.518,A -85,B 0,C 180,E1 21634.189,E2 21634.189} C_VEL
LIN {X 0,Y 441.156,Z 307.527,A -85,B 0,C 180,E1 21630.51,E2 21630.51} C_VEL
LIN {X 0,Y 441.148,Z 307.532,A -85,B 0,C 180,E1 21626.81,E2 21626.81} C_VEL
LIN {X 0,Y 441.151,Z 307.533,A -85,B 0,C 180,E1 21623.05,E2 21623.05} C_VEL
LIN {X 0,Y 441.175,Z 307.513,A -85,B 0,C 180,E1 21619.461,E2 21619.461} C_VEL
LIN {X 0,Y 441.184,Z 307.523,A -85,B 0,C 180,E1 21615.781,E2 21615.781} C_VEL
LIN {X 0,Y 441.144,Z 307.529,A -85,B 0,C 180,E1 21612.169,E2 21612.169} C_VEL
LIN {X 0,Y 441.126,Z 307.513,A -85,B 0,C 180,E1 21608.472,E2 21608.472} C_VEL
LIN {X 0,Y 441.123,Z 307.531,A -85,B 0,C 180,E1 21604.681,E2 21604.681} C_VEL
LIN {X 0,Y 441.137,Z 307.533,A -85,B 0,C 180,E1 21601.039,E2 21601.039} C_VEL
LIN {X 0,Y 441.166,Z 307.512,A -85,B 0,C 180,E1 21597.402,E2 21597.402} C_VEL
LIN {X 0,Y 441.167,Z 307.528,A -85,B 0,C 180,E1 21593.624,E2 21593.624} C_VEL
LIN {X 0,Y 441.141,Z 307.529,A -85,B 0,C 180,E1 21589.949,E2 21589.949} C_VEL
LIN {X 0,Y 441.132,Z 307.515,A -85,B 0,C 180,E1 21586.232,E2 21586.232} C_VEL
LIN {X 0,Y 441.136,Z 307.526,A -85,B 0,C 180,E1 21582.455,E2 21582.455} C_VEL
LIN {X 0,Y 441.155,Z 307.53,A -85,B 0,C 180,E1 21578.738,E2 21578.738} C_VEL
LIN {X 0,Y 441.188,Z 307.531,A -85,B 0,C 180,E1 21575.069,E2 21575.069} C_VEL
LIN {X 0,Y 441.203,Z 307.527,A -85,B 0,C 180,E1 21571.282,E2 21571.282} C_VEL
LIN {X 0,Y 441.177,Z 307.53,A -85,B 0,C 180,E1 21567.512,E2 21567.512} C_VEL
LIN {X 0,Y 441.158,Z 307.485,A -85,B 0,C 180,E1 21563.787,E2 21563.787} C_VEL
LIN {X 0,Y 441.158,Z 307.518,A -85,B 0,C 180,E1 21560.104,E2 21560.104} C_VEL
LIN {X 0,Y 441.172,Z 307.517,A -85,B 0,C 180,E1 21556.451,E2 21556.451} C_VEL
LIN {X 0,Y 441.225,Z 307.774,A -85,B 0,C 180,E1 21555.36,E2 21555.36} C_VEL
LIN {X 0,Y 442.653,Z 311.217,A -85,B 0,C 180,E1 21554.826,E2 21554.826} C_VEL
LIN {X 0,Y 451.265,Z 330.255,A -85,B 0,C 180,E1 21552.266,E2 21552.266} C_VEL
LIN {X 0,Y 459.55,Z 350.659,A -85,B 0,C 180,E1 21549.823,E2 21549.823} C_VEL
LIN {X 0,Y 460.574,Z 353.601,A -85,B 0,C 180,E1 21549.498,E2 21549.498} C_VEL
LIN {X 0,Y 458.278,Z 385.51,A -85,B 0,C 180,E1 21547.218,E2 21547.218} C_VEL
LIN {X 0,Y 461.594,Z 416.023,A -85,B 0,C 180,E1 21546.357,E2 21546.357} C_VEL
LIN {X 0,Y 456.582,Z 638.411,A -85,B 0,C 180,E1 21542.453,E2 21542.453} C_VEL
LIN {X 0,Y 455.51,Z 660.4,A -85,B 0,C 180,E1 21541.896,E2 21541.896} C_VEL
LIN {X 0,Y 454.066,Z 681.451,A -85,B 0,C 180,E1 21541.125,E2 21541.125} C_VEL
LIN {X 0,Y 452.521,Z 701.039,A -85,B 0,C 180,E1 21540.176,E2 21540.176} C_VEL
LIN {X 0,Y 450.788,Z 720.778,A -85,B 0,C 180,E1 21538.972,E2 21538.972} C_VEL
LIN {X 0,Y 448.957,Z 740.152,A -85,B 0,C 180,E1 21537.523,E2 21537.523} C_VEL
LIN {X 0,Y 447.195,Z 758.68,A -85,B 0,C 180,E1 21535.847,E2 21535.847} C_VEL
LIN {X 0,Y 445.465,Z 776.639,A -85,B 0,C 180,E1 21533.91,E2 21533.91} C_VEL
LIN {X 0,Y 443.924,Z 793.523,A -85,B 0,C 180,E1 21531.746,E2 21531.746} C_VEL
LIN {X 0,Y 442.7,Z 808.087,A -85,B 0,C 180,E1 21529.527,E2 21529.527} C_VEL
LIN {X 0,Y 441.739,Z 820.649,A -85,B 0,C 180,E1 21527.248,E2 21527.248} C_VEL
LIN {X 0,Y 441.072,Z 831.137,A -85,B 0,C 180,E1 21524.976,E2 21524.976} C_VEL
LIN {X 0,Y 440.59,Z 840.306,A -85,B 0,C 180,E1 21522.583,E2 21522.583} C_VEL
LIN {X 0,Y 440.322,Z 847.692,A -85,B 0,C 180,E1 21520.202,E2 21520.202} C_VEL
LIN {X 0,Y 440.193,Z 853.586,A -85,B 0,C 180,E1 21517.701,E2 21517.701} C_VEL
LIN {X 0,Y 440.159,Z 857.778,A -85,B 0,C 180,E1 21515.213,E2 21515.213} C_VEL
LIN {X 0,Y 440.166,Z 860.368,A -85,B 0,C 180,E1 21512.734,E2 21512.734} C_VEL
LIN {X 0,Y 440.17,Z 861.323,A -85,B 0,C 180,E1 21510.26,E2 21510.26} C_VEL
LIN {X 0,Y 440.163,Z 860.669,A -85,B 0,C 180,E1 21507.787,E2 21507.787} C_VEL
LIN {X 0,Y 440.152,Z 858.475,A -85,B 0,C 180,E1 21505.309,E2 21505.309} C_VEL
LIN {X 0,Y 440.18,Z 854.64,A -85,B 0,C 180,E1 21502.823,E2 21502.823} C_VEL
LIN {X 0,Y 440.299,Z 849.047,A -85,B 0,C 180,E1 21500.326,E2 21500.326} C_VEL
LIN {X 0,Y 440.536,Z 841.653,A -85,B 0,C 180,E1 21497.815,E2 21497.815} C_VEL
LIN {X 0,Y 440.979,Z 832.844,A -85,B 0,C 180,E1 21495.424,E2 21495.424} C_VEL
LIN {X 0,Y 441.647,Z 822.041,A -85,B 0,C 180,E1 21493.02,E2 21493.02} C_VEL
LIN {X 0,Y 442.571,Z 809.682,A -85,B 0,C 180,E1 21490.741,E2 21490.741} C_VEL
LIN {X 0,Y 443.709,Z 795.842,A -85,B 0,C 180,E1 21488.59,E2 21488.59} C_VEL
LIN {X 0,Y 445.087,Z 780.574,A -85,B 0,C 180,E1 21486.571,E2 21486.571} C_VEL
LIN {X 0,Y 446.736,Z 763.246,A -85,B 0,C 180,E1 21484.622,E2 21484.622} C_VEL
LIN {X 0,Y 448.509,Z 744.809,A -85,B 0,C 180,E1 21482.879,E2 21482.879} C_VEL
LIN {X 0,Y 450.297,Z 726.014,A -85,B 0,C 180,E1 21481.398,E2 21481.398} C_VEL
LIN {X 0,Y 452.02,Z 706.85,A -85,B 0,C 180,E1 21480.153,E2 21480.153} C_VEL
LIN {X 0,Y 453.682,Z 686.699,A -85,B 0,C 180,E1 21479.104,E2 21479.104} C_VEL
LIN {X 0,Y 455.181,Z 665.713,A -85,B 0,C 180,E1 21478.269,E2 21478.269} C_VEL
LIN {X 0,Y 456.417,Z 643.585,A -85,B 0,C 180,E1 21477.652,E2 21477.652} C_VEL
LIN {X 0,Y 461.361,Z 425.998,A -85,B 0,C 180,E1 21473.816,E2 21473.816} C_VEL
LIN {X 0,Y 461.425,Z 412.906,A -85,B 0,C 180,E1 21473.572,E2 21473.572} C_VEL
LIN {X 0,Y 458.225,Z 384.258,A -85,B 0,C 180,E1 21472.727,E2 21472.727} C_VEL
LIN {X 0,Y 460.497,Z 353.204,A -85,B 0,C 180,E1 21470.469,E2 21470.469} C_VEL
LIN {X 0,Y 452.108,Z 332.26,A -85,B 0,C 180,E1 21467.994,E2 21467.994} C_VEL
LIN {X 0,Y 444.308,Z 314.885,A -85,B 0,C 180,E1 21465.694,E2 21465.694} C_VEL
LIN {X 0,Y 441.262,Z 307.966,A -85,B 0,C 180,E1 21464.704,E2 21464.704} C_VEL
LIN {X 0,Y 441.179,Z 307.533,A -85,B 0,C 180,E1 21464.449,E2 21464.449} C_VEL
LIN {X 0,Y 441.197,Z 307.494,A -85,B 0,C 180,E1 21460.743,E2 21460.743} C_VEL
LIN {X 0,Y 441.19,Z 307.49,A -85,B 0,C 180,E1 21457.072,E2 21457.072} C_VEL
LIN {X 0,Y 441.167,Z 307.529,A -85,B 0,C 180,E1 21453.417,E2 21453.417} C_VEL
LIN {X 0,Y 441.151,Z 307.533,A -85,B 0,C 180,E1 21449.759,E2 21449.759} C_VEL
LIN {X 0,Y 441.155,Z 307.531,A -85,B 0,C 180,E1 21446.084,E2 21446.084} C_VEL
LIN {X 0,Y 441.172,Z 307.521,A -85,B 0,C 180,E1 21442.38,E2 21442.38} C_VEL
LIN {X 0,Y 441.188,Z 307.515,A -85,B 0,C 180,E1 21438.635,E2 21438.635} C_VEL
LIN {X 0,Y 441.179,Z 307.523,A -85,B 0,C 180,E1 21434.838,E2 21434.838} C_VEL
LIN {X 0,Y 441.149,Z 307.531,A -85,B 0,C 180,E1 21431.107,E2 21431.107} C_VEL
LIN {X 0,Y 441.129,Z 307.523,A -85,B 0,C 180,E1 21427.423,E2 21427.423} C_VEL
LIN {X 0,Y 441.123,Z 307.523,A -85,B 0,C 180,E1 21423.638,E2 21423.638} C_VEL
LIN {X 0,Y 441.138,Z 307.535,A -85,B 0,C 180,E1 21420,E2 21420} C_VEL
LIN {X 0,Y 441.164,Z 307.515,A -85,B 0,C 180,E1 21416.361,E2 21416.361} C_VEL
LIN {X 0,Y 441.166,Z 307.519,A -85,B 0,C 180,E1 21412.577,E2 21412.577} C_VEL
LIN {X 0,Y 441.141,Z 307.533,A -85,B 0,C 180,E1 21408.892,E2 21408.892} C_VEL
LIN {X 0,Y 441.129,Z 307.517,A -85,B 0,C 180,E1 21405.294,E2 21405.294} C_VEL
LIN {X 0,Y 441.137,Z 307.525,A -85,B 0,C 180,E1 21401.499,E2 21401.499} C_VEL
LIN {X 0,Y 441.166,Z 307.531,A -85,B 0,C 180,E1 21397.9,E2 21397.9} C_VEL
LIN {X 0,Y 441.188,Z 307.518,A -85,B 0,C 180,E1 21394.206,E2 21394.206} C_VEL
LIN {X 0,Y 441.175,Z 307.517,A -85,B 0,C 180,E1 21390.488,E2 21390.488} C_VEL
LIN {X 0,Y 441.151,Z 307.527,A -85,B 0,C 180,E1 21386.892,E2 21386.892} C_VEL
LIN {X 0,Y 441.152,Z 307.532,A -85,B 0,C 180,E1 21383.086,E2 21383.086} C_VEL
LIN {X 0,Y 441.166,Z 307.528,A -85,B 0,C 180,E1 21379.396,E2 21379.396} C_VEL
LIN {X 0,Y 441.189,Z 307.518,A -85,B 0,C 180,E1 21375.732,E2 21375.732} C_VEL
LIN {X 0,Y 441.199,Z 307.512,A -85,B 0,C 180,E1 21371.953,E2 21371.953} C_VEL
LIN {X 0,Y 441.194,Z 307.492,A -85,B 0,C 180,E1 21368.15,E2 21368.15} C_VEL
LIN {X 0,Y 441.209,Z 307.82,A -85,B 0,C 180,E1 21367.029,E2 21367.029} C_VEL
LIN {X 0,Y 447.654,Z 324.815,A -85,B 0,C 180,E1 21364.153,E2 21364.153} C_VEL
LIN {X 0,Y 453.387,Z 341.24,A -85,B 0,C 180,E1 21361.651,E2 21361.651} C_VEL
LIN {X 0,Y 457.468,Z 349.456,A -85,B 0,C 180,E1 21361.119,E2 21361.119} C_VEL
LIN {X 0,Y 460.259,Z 363.748,A -85,B 0,C 180,E1 21360.631,E2 21360.631} C_VEL
LIN {X 0,Y 458.427,Z 485.244,A -85,B 0,C 180,E1 21358.751,E2 21358.751} C_VEL
LIN {X 0,Y 457.493,Z 492.941,A -85,B 0,C 180,E1 21358.699,E2 21358.699} C_VEL
LIN {X 0,Y 451.905,Z 513.429,A -85,B 0,C 180,E1 21358.802,E2 21358.802} C_VEL
LIN {X 0,Y 451.164,Z 520.038,A -85,B 0,C 180,E1 21358.752,E2 21358.752} C_VEL
LIN {X 0,Y 450.675,Z 558.225,A -85,B 0,C 180,E1 21358.114,E2 21358.114} C_VEL
LIN {X 0,Y 450.095,Z 576.922,A -85,B 0,C 180,E1 21357.568,E2 21357.568} C_VEL
LIN {X 0,Y 449.101,Z 595.146,A -85,B 0,C 180,E1 21356.797,E2 21356.797} C_VEL
LIN {X 0,Y 447.783,Z 612.586,A -85,B 0,C 180,E1 21355.811,E2 21355.811} C_VEL
LIN {X 0,Y 446.132,Z 629.477,A -85,B 0,C 180,E1 21354.596,E2 21354.596} C_VEL
LIN {X 0,Y 444.321,Z 645.19,A -85,B 0,C 180,E1 21353.191,E2 21353.191} C_VEL
LIN {X 0,Y 442.435,Z 659.626,A -85,B 0,C 180,E1 21351.614,E2 21351.614} C_VEL
LIN {X 0,Y 440.617,Z 672.62,A -85,B 0,C 180,E1 21349.9,E2 21349.9} C_VEL
LIN {X 0,Y 438.761,Z 685.034,A -85,B 0,C 180,E1 21347.917,E2 21347.917} C_VEL
LIN {X 0,Y 437.134,Z 695.913,A -85,B 0,C 180,E1 21345.794,E2 21345.794} C_VEL
LIN {X 0,Y 435.747,Z 705.314,A -85,B 0,C 180,E1 21343.535,E2 21343.535} C_VEL
LIN {X 0,Y 434.648,Z 713.225,A -85,B 0,C 180,E1 21341.141,E2 21341.141} C_VEL
LIN {X 0,Y 433.863,Z 719.607,A -85,B 0,C 180,E1 21338.615,E2 21338.615} C_VEL
LIN {X 0,Y 433.335,Z 724.297,A -85,B 0,C 180,E1 21336.025,E2 21336.025} C_VEL
LIN {X 0,Y 433.043,Z 727.257,A -85,B 0,C 180,E1 21333.442,E2 21333.442} C_VEL
LIN {X 0,Y 432.935,Z 728.607,A -85,B 0,C 180,E1 21330.794,E2 21330.794} C_VEL
LIN {X 0,Y 432.96,Z 728.305,A -85,B 0,C 180,E1 21328.147,E2 21328.147} C_VEL
LIN {X 0,Y 433.131,Z 726.337,A -85,B 0,C 180,E1 21325.499,E2 21325.499} C_VEL
LIN {X 0,Y 433.513,Z 722.623,A -85,B 0,C 180,E1 21322.846,E2 21322.846} C_VEL
LIN {X 0,Y 434.128,Z 717.343,A -85,B 0,C 180,E1 21320.316,E2 21320.316} C_VEL
LIN {X 0,Y 435.05,Z 710.224,A -85,B 0,C 180,E1 21317.794,E2 21317.794} C_VEL
LIN {X 0,Y 436.226,Z 702.029,A -85,B 0,C 180,E1 21315.533,E2 21315.533} C_VEL
LIN {X 0,Y 437.631,Z 692.499,A -85,B 0,C 180,E1 21313.406,E2 21313.406} C_VEL
LIN {X 0,Y 439.261,Z 681.655,A -85,B 0,C 180,E1 21311.418,E2 21311.418} C_VEL
LIN {X 0,Y 441.063,Z 669.469,A -85,B 0,C 180,E1 21309.568,E2 21309.568} C_VEL
LIN {X 0,Y 443.026,Z 655.276,A -85,B 0,C 180,E1 21307.789,E2 21307.789} C_VEL
LIN {X 0,Y 444.968,Z 639.901,A -85,B 0,C 180,E1 21306.213,E2 21306.213} C_VEL
LIN {X 0,Y 446.682,Z 624.188,A -85,B 0,C 180,E1 21304.902,E2 21304.902} C_VEL
LIN {X 0,Y 448.259,Z 606.922,A -85,B 0,C 180,E1 21303.75,E2 21303.75} C_VEL
LIN {X 0,Y 449.453,Z 589.653,A -85,B 0,C 180,E1 21302.855,E2 21302.855} C_VEL
LIN {X 0,Y 450.342,Z 570.833,A -85,B 0,C 180,E1 21302.138,E2 21302.138} C_VEL
LIN {X 0,Y 450.77,Z 551.683,A -85,B 0,C 180,E1 21301.658,E2 21301.658} C_VEL
LIN {X 0,Y 453.513,Z 363.494,A -85,B 0,C 180,E1 21298.685,E2 21298.685} C_VEL
LIN {X 0,Y 450.831,Z 351.762,A -85,B 0,C 180,E1 21298.24,E2 21298.24} C_VEL
LIN {X 0,Y 445.523,Z 341.845,A -85,B 0,C 180,E1 21297.548,E2 21297.548} C_VEL
LIN {X 0,Y 439.445,Z 324.714,A -85,B 0,C 180,E1 21294.856,E2 21294.856} C_VEL
LIN {X 0,Y 433.917,Z 310.839,A -85,B 0,C 180,E1 21292.436,E2 21292.436} C_VEL
LIN {X 0,Y 433.292,Z 308.724,A -85,B 0,C 180,E1 21292.037,E2 21292.037} C_VEL
LIN {X 0,Y 433.254,Z 308.51,A -85,B 0,C 180,E1 21288.347,E2 21288.347} C_VEL
LIN {X 0,Y 433.238,Z 308.496,A -85,B 0,C 180,E1 21284.511,E2 21284.511} C_VEL
LIN {X 0,Y 433.222,Z 308.514,A -85,B 0,C 180,E1 21280.78,E2 21280.78} C_VEL
LIN {X 0,Y 433.22,Z 308.515,A -85,B 0,C 180,E1 21277.01,E2 21277.01} C_VEL
LIN {X 0,Y 433.228,Z 308.509,A -85,B 0,C 180,E1 21273.318,E2 21273.318} C_VEL
LIN {X 0,Y 433.251,Z 308.503,A -85,B 0,C 180,E1 21269.596,E2 21269.596} C_VEL
LIN {X 0,Y 433.252,Z 308.508,A -85,B 0,C 180,E1 21265.84,E2 21265.84} C_VEL
LIN {X 0,Y 433.231,Z 308.52,A -85,B 0,C 180,E1 21262.098,E2 21262.098} C_VEL
LIN {X 0,Y 433.205,Z 308.513,A -85,B 0,C 180,E1 21258.434,E2 21258.434} C_VEL
LIN {X 0,Y 433.195,Z 308.504,A -85,B 0,C 180,E1 21254.708,E2 21254.708} C_VEL
LIN {X 0,Y 433.198,Z 308.52,A -85,B 0,C 180,E1 21250.91,E2 21250.91} C_VEL
LIN {X 0,Y 433.22,Z 308.51,A -85,B 0,C 180,E1 21247.293,E2 21247.293} C_VEL
LIN {X 0,Y 433.229,Z 308.502,A -85,B 0,C 180,E1 21243.573,E2 21243.573} C_VEL
LIN {X 0,Y 433.204,Z 308.523,A -85,B 0,C 180,E1 21239.868,E2 21239.868} C_VEL
LIN {X 0,Y 433.186,Z 308.511,A -85,B 0,C 180,E1 21236.162,E2 21236.162} C_VEL
LIN {X 0,Y 433.185,Z 308.509,A -85,B 0,C 180,E1 21232.44,E2 21232.44} C_VEL
LIN {X 0,Y 433.199,Z 308.521,A -85,B 0,C 180,E1 21228.686,E2 21228.686} C_VEL
LIN {X 0,Y 433.226,Z 308.516,A -85,B 0,C 180,E1 21225.02,E2 21225.02} C_VEL
LIN {X 0,Y 433.248,Z 308.503,A -85,B 0,C 180,E1 21221.29,E2 21221.29} C_VEL
LIN {X 0,Y 433.243,Z 308.506,A -85,B 0,C 180,E1 21217.474,E2 21217.474} C_VEL
LIN {X 0,Y 433.217,Z 308.517,A -85,B 0,C 180,E1 21213.844,E2 21213.844} C_VEL
LIN {X 0,Y 433.211,Z 308.521,A -85,B 0,C 180,E1 21210.203,E2 21210.203} C_VEL
LIN {X 0,Y 433.219,Z 308.518,A -85,B 0,C 180,E1 21206.424,E2 21206.424} C_VEL
LIN {X 0,Y 433.241,Z 308.48,A -85,B 0,C 180,E1 21202.768,E2 21202.768} C_VEL
LIN {X 0,Y 433.261,Z 308.478,A -85,B 0,C 180,E1 21199.05,E2 21199.05} C_VEL
LIN {X 0,Y 433.246,Z 308.659,A -85,B 0,C 180,E1 21196.247,E2 21196.247} C_VEL
LIN {X 0,Y 433.614,Z 310.179,A -85,B 0,C 180,E1 21195.965,E2 21195.965} C_VEL
LIN {X 0,Y 437.237,Z 317.665,A -85,B 0,C 180,E1 21194.855,E2 21194.855} C_VEL
LIN {X 0,Y 445.378,Z 335.804,A -85,B 0,C 180,E1 21192.389,E2 21192.389} C_VEL
LIN {X 0,Y 453.62,Z 356.435,A -85,B 0,C 180,E1 21189.888,E2 21189.888} C_VEL
LIN {X 0,Y 451.434,Z 385.093,A -85,B 0,C 180,E1 21187.81,E2 21187.81} C_VEL
LIN {X 0,Y 454.866,Z 417.183,A -85,B 0,C 180,E1 21186.886,E2 21186.886} C_VEL
LIN {X 0,Y 449.594,Z 637.692,A -85,B 0,C 180,E1 21182.957,E2 21182.957} C_VEL
LIN {X 0,Y 448.473,Z 659.52,A -85,B 0,C 180,E1 21182.395,E2 21182.395} C_VEL
LIN {X 0,Y 446.911,Z 680.761,A -85,B 0,C 180,E1 21181.605,E2 21181.605} C_VEL
LIN {X 0,Y 445.281,Z 700.245,A -85,B 0,C 180,E1 21180.644,E2 21180.644} C_VEL
LIN {X 0,Y 443.452,Z 719.693,A -85,B 0,C 180,E1 21179.44,E2 21179.44} C_VEL
LIN {X 0,Y 441.492,Z 739.191,A -85,B 0,C 180,E1 21177.955,E2 21177.955} C_VEL
LIN {X 0,Y 439.603,Z 757.767,A -85,B 0,C 180,E1 21176.243,E2 21176.243} C_VEL
LIN {X 0,Y 437.756,Z 775.628,A -85,B 0,C 180,E1 21174.275,E2 21174.275} C_VEL
LIN {X 0,Y 436.179,Z 791.723,A -85,B 0,C 180,E1 21172.167,E2 21172.167} C_VEL
LIN {X 0,Y 434.853,Z 806.474,A -85,B 0,C 180,E1 21169.879,E2 21169.879} C_VEL
LIN {X 0,Y 433.845,Z 819.048,A -85,B 0,C 180,E1 21167.572,E2 21167.572} C_VEL
LIN {X 0,Y 433.139,Z 829.782,A -85,B 0,C 180,E1 21165.224,E2 21165.224} C_VEL
LIN {X 0,Y 432.642,Z 839.047,A -85,B 0,C 180,E1 21162.771,E2 21162.771} C_VEL
LIN {X 0,Y 432.381,Z 846.347,A -85,B 0,C 180,E1 21160.391,E2 21160.391} C_VEL
LIN {X 0,Y 432.255,Z 852.295,A -85,B 0,C 180,E1 21157.844,E2 21157.844} C_VEL
LIN {X 0,Y 432.237,Z 856.537,A -85,B 0,C 180,E1 21155.309,E2 21155.309} C_VEL
LIN {X 0,Y 432.253,Z 859.158,A -85,B 0,C 180,E1 21152.784,E2 21152.784} C_VEL
LIN {X 0,Y 432.26,Z 860.121,A -85,B 0,C 180,E1 21150.265,E2 21150.265} C_VEL
LIN {X 0,Y 432.25,Z 859.462,A -85,B 0,C 180,E1 21147.746,E2 21147.746} C_VEL
LIN {X 0,Y 432.232,Z 857.242,A -85,B 0,C 180,E1 21145.223,E2 21145.223} C_VEL
LIN {X 0,Y 432.24,Z 853.371,A -85,B 0,C 180,E1 21142.691,E2 21142.691} C_VEL
LIN {X 0,Y 432.348,Z 847.66,A -85,B 0,C 180,E1 21140.122,E2 21140.122} C_VEL
LIN {X 0,Y 432.588,Z 840.256,A -85,B 0,C 180,E1 21137.587,E2 21137.587} C_VEL
LIN {X 0,Y 433.08,Z 830.793,A -85,B 0,C 180,E1 21135.015,E2 21135.015} C_VEL
LIN {X 0,Y 433.785,Z 819.943,A -85,B 0,C 180,E1 21132.602,E2 21132.602} C_VEL
LIN {X 0,Y 434.795,Z 807.228,A -85,B 0,C 180,E1 21130.243,E2 21130.243} C_VEL
LIN {X 0,Y 436.125,Z 792.314,A -85,B 0,C 180,E1 21127.915,E2 21127.915} C_VEL
LIN {X 0,Y 437.756,Z 775.626,A -85,B 0,C 180,E1 21125.725,E2 21125.725} C_VEL
LIN {X 0,Y 439.603,Z 757.758,A -85,B 0,C 180,E1 21123.756,E2 21123.756} C_VEL
LIN {X 0,Y 441.51,Z 739.029,A -85,B 0,C 180,E1 21122.031,E2 21122.031} C_VEL
LIN {X 0,Y 443.451,Z 719.67,A -85,B 0,C 180,E1 21120.56,E2 21120.56} C_VEL
LIN {X 0,Y 445.278,Z 700.21,A -85,B 0,C 180,E1 21119.356,E2 21119.356} C_VEL
LIN {X 0,Y 446.967,Z 679.972,A -85,B 0,C 180,E1 21118.361,E2 21118.361} C_VEL
LIN {X 0,Y 448.497,Z 659.076,A -85,B 0,C 180,E1 21117.593,E2 21117.593} C_VEL
LIN {X 0,Y 449.61,Z 636.961,A -85,B 0,C 180,E1 21117.03,E2 21117.03} C_VEL
LIN {X 0,Y 454.893,Z 415.647,A -85,B 0,C 180,E1 21113.089,E2 21113.089} C_VEL
LIN {X 0,Y 451.359,Z 384.026,A -85,B 0,C 180,E1 21112.15,E2 21112.15} C_VEL
LIN {X 0,Y 453.541,Z 356.253,A -85,B 0,C 180,E1 21110.096,E2 21110.096} C_VEL
LIN {X 0,Y 445.35,Z 335.77,A -85,B 0,C 180,E1 21107.615,E2 21107.615} C_VEL
LIN {X 0,Y 437.614,Z 318.561,A -85,B 0,C 180,E1 21105.281,E2 21105.281} C_VEL
LIN {X 0,Y 434.4,Z 311.792,A -85,B 0,C 180,E1 21104.291,E2 21104.291} C_VEL
LIN {X 0,Y 433.262,Z 308.771,A -85,B 0,C 180,E1 21103.814,E2 21103.814} C_VEL
LIN {X 0,Y 433.249,Z 308.485,A -85,B 0,C 180,E1 21100.602,E2 21100.602} C_VEL
LIN {X 0,Y 433.256,Z 308.473,A -85,B 0,C 180,E1 21096.871,E2 21096.871} C_VEL
LIN {X 0,Y 433.256,Z 308.517,A -85,B 0,C 180,E1 21092.999,E2 21092.999} C_VEL
LIN {X 0,Y 433.232,Z 308.521,A -85,B 0,C 180,E1 21089.266,E2 21089.266} C_VEL
LIN {X 0,Y 433.213,Z 308.522,A -85,B 0,C 180,E1 21085.524,E2 21085.524} C_VEL
LIN {X 0,Y 433.205,Z 308.52,A -85,B 0,C 180,E1 21081.814,E2 21081.814} C_VEL
LIN {X 0,Y 433.215,Z 308.507,A -85,B 0,C 180,E1 21078.154,E2 21078.154} C_VEL
LIN {X 0,Y 433.237,Z 308.504,A -85,B 0,C 180,E1 21074.433,E2 21074.433} C_VEL
LIN {X 0,Y 433.241,Z 308.521,A -85,B 0,C 180,E1 21070.639,E2 21070.639} C_VEL
LIN {X 0,Y 433.218,Z 308.511,A -85,B 0,C 180,E1 21066.893,E2 21066.893} C_VEL
LIN {X 0,Y 433.192,Z 308.507,A -85,B 0,C 180,E1 21063.175,E2 21063.175} C_VEL
LIN {X 0,Y 433.181,Z 308.524,A -85,B 0,C 180,E1 21059.471,E2 21059.471} C_VEL
LIN {X 0,Y 433.182,Z 308.52,A -85,B 0,C 180,E1 21055.631,E2 21055.631} C_VEL
LIN {X 0,Y 433.201,Z 308.502,A -85,B 0,C 180,E1 21051.945,E2 21051.945} C_VEL
LIN {X 0,Y 433.236,Z 308.52,A -85,B 0,C 180,E1 21048.282,E2 21048.282} C_VEL
LIN {X 0,Y 433.239,Z 308.506,A -85,B 0,C 180,E1 21044.472,E2 21044.472} C_VEL
LIN {X 0,Y 433.215,Z 308.505,A -85,B 0,C 180,E1 21040.725,E2 21040.725} C_VEL
LIN {X 0,Y 433.203,Z 308.522,A -85,B 0,C 180,E1 21037.041,E2 21037.041} C_VEL
LIN {X 0,Y 433.204,Z 308.521,A -85,B 0,C 180,E1 21033.251,E2 21033.251} C_VEL
LIN {X 0,Y 433.214,Z 308.515,A -85,B 0,C 180,E1 21029.485,E2 21029.485} C_VEL
LIN {X 0,Y 433.246,Z 308.506,A -85,B 0,C 180,E1 21025.888,E2 21025.888} C_VEL
LIN {X 0,Y 433.261,Z 308.506,A -85,B 0,C 180,E1 21022.113,E2 21022.113} C_VEL
LIN {X 0,Y 433.247,Z 308.508,A -85,B 0,C 180,E1 21018.344,E2 21018.344} C_VEL
LIN {X 0,Y 433.23,Z 308.48,A -85,B 0,C 180,E1 21014.554,E2 21014.554} C_VEL
LIN {X 0,Y 433.224,Z 308.523,A -85,B 0,C 180,E1 21010.778,E2 21010.778} C_VEL
LIN {X 0,Y 433.288,Z 308.703,A -85,B 0,C 180,E1 21007.865,E2 21007.865} C_VEL
LIN {X 0,Y 439.62,Z 325.147,A -85,B 0,C 180,E1 21004.968,E2 21004.968} C_VEL
LIN {X 0,Y 445.697,Z 342.303,A -85,B 0,C 180,E1 21002.308,E2 21002.308} C_VEL
LIN {X 0,Y 451.327,Z 353.188,A -85,B 0,C 180,E1 21001.59,E2 21001.59} C_VEL
LIN {X 0,Y 453.612,Z 365.256,A -85,B 0,C 180,E1 21001.173,E2 21001.173} C_VEL
LIN {X 0,Y 451.164,Z 520.038,A -85,B 0,C 180,E1 20998.752,E2 20998.752} C_VEL
LIN {X 0,Y 450.198,Z 527.737,A -85,B 0,C 180,E1 20998.703,E2 20998.703} C_VEL
LIN {X 0,Y 444.61,Z 548.211,A -85,B 0,C 180,E1 20998.805,E2 20998.805} C_VEL
LIN {X 0,Y 443.897,Z 554.794,A -85,B 0,C 180,E1 20998.73,E2 20998.73} C_VEL
LIN {X 0,Y 443.414,Z 573.367,A -85,B 0,C 180,E1 20998.233,E2 20998.233} C_VEL
LIN {X 0,Y 442.477,Z 591.376,A -85,B 0,C 180,E1 20997.522,E2 20997.522} C_VEL
LIN {X 0,Y 441.192,Z 608.876,A -85,B 0,C 180,E1 20996.588,E2 20996.588} C_VEL
LIN {X 0,Y 439.554,Z 625.744,A -85,B 0,C 180,E1 20995.436,E2 20995.436} C_VEL
LIN {X 0,Y 437.703,Z 641.812,A -85,B 0,C 180,E1 20994.063,E2 20994.063} C_VEL
LIN {X 0,Y 435.672,Z 657.035,A -85,B 0,C 180,E1 20992.464,E2 20992.464} C_VEL
LIN {X 0,Y 433.613,Z 671.113,A -85,B 0,C 180,E1 20990.658,E2 20990.658} C_VEL
LIN {X 0,Y 431.721,Z 683.211,A -85,B 0,C 180,E1 20988.779,E2 20988.779} C_VEL
LIN {X 0,Y 429.901,Z 694.651,A -85,B 0,C 180,E1 20986.619,E2 20986.619} C_VEL
LIN {X 0,Y 428.36,Z 704.508,A -85,B 0,C 180,E1 20984.325,E2 20984.325} C_VEL
LIN {X 0,Y 427.097,Z 712.854,A -85,B 0,C 180,E1 20981.888,E2 20981.888} C_VEL
LIN {X 0,Y 426.22,Z 719.323,A -85,B 0,C 180,E1 20979.451,E2 20979.451} C_VEL
LIN {X 0,Y 425.589,Z 724.368,A -85,B 0,C 180,E1 20976.881,E2 20976.881} C_VEL
LIN {X 0,Y 425.222,Z 727.728,A -85,B 0,C 180,E1 20974.315,E2 20974.315} C_VEL
LIN {X 0,Y 425.048,Z 729.585,A -85,B 0,C 180,E1 20971.618,E2 20971.618} C_VEL
LIN {X 0,Y 425.026,Z 729.784,A -85,B 0,C 180,E1 20968.922,E2 20968.922} C_VEL
LIN {X 0,Y 425.165,Z 728.333,A -85,B 0,C 180,E1 20966.225,E2 20966.225} C_VEL
LIN {X 0,Y 425.506,Z 725.175,A -85,B 0,C 180,E1 20963.524,E2 20963.524} C_VEL
LIN {X 0,Y 426.124,Z 720.184,A -85,B 0,C 180,E1 20960.819,E2 20960.819} C_VEL
LIN {X 0,Y 427.01,Z 713.565,A -85,B 0,C 180,E1 20958.246,E2 20958.246} C_VEL
LIN {X 0,Y 428.236,Z 705.404,A -85,B 0,C 180,E1 20955.809,E2 20955.809} C_VEL
LIN {X 0,Y 429.75,Z 695.733,A -85,B 0,C 180,E1 20953.511,E2 20953.511} C_VEL
LIN {X 0,Y 431.529,Z 684.545,A -85,B 0,C 180,E1 20951.353,E2 20951.353} C_VEL
LIN {X 0,Y 433.398,Z 672.724,A -85,B 0,C 180,E1 20949.473,E2 20949.473} C_VEL
LIN {X 0,Y 435.425,Z 658.978,A -85,B 0,C 180,E1 20947.665,E2 20947.665} C_VEL
LIN {X 0,Y 437.429,Z 644.175,A -85,B 0,C 180,E1 20946.064,E2 20946.064} C_VEL
LIN {X 0,Y 439.316,Z 628.345,A -85,B 0,C 180,E1 20944.668,E2 20944.668} C_VEL
LIN {X 0,Y 441.008,Z 611.462,A -85,B 0,C 180,E1 20943.472,E2 20943.472} C_VEL
LIN {X 0,Y 442.353,Z 594.052,A -85,B 0,C 180,E1 20942.506,E2 20942.506} C_VEL
LIN {X 0,Y 443.357,Z 575.671,A -85,B 0,C 180,E1 20941.747,E2 20941.747} C_VEL
LIN {X 0,Y 443.911,Z 556.954,A -85,B 0,C 180,E1 20941.219,E2 20941.219} C_VEL
LIN {X 0,Y 446.899,Z 364.901,A -85,B 0,C 180,E1 20938.123,E2 20938.123} C_VEL
LIN {X 0,Y 444.689,Z 355.34,A -85,B 0,C 180,E1 20937.747,E2 20937.747} C_VEL
LIN {X 0,Y 437.741,Z 342.648,A -85,B 0,C 180,E1 20936.839,E2 20936.839} C_VEL
LIN {X 0,Y 431.644,Z 325.832,A -85,B 0,C 180,E1 20934.124,E2 20934.124} C_VEL
LIN {X 0,Y 426.384,Z 312.582,A -85,B 0,C 180,E1 20931.753,E2 20931.753} C_VEL
LIN {X 0,Y 425.328,Z 309.748,A -85,B 0,C 180,E1 20931.195,E2 20931.195} C_VEL
LIN {X 0,Y 425.313,Z 309.498,A -85,B 0,C 180,E1 20928.382,E2 20928.382} C_VEL
LIN {X 0,Y 425.295,Z 309.481,A -85,B 0,C 180,E1 20924.576,E2 20924.576} C_VEL
LIN {X 0,Y 425.284,Z 309.502,A -85,B 0,C 180,E1 20920.799,E2 20920.799} C_VEL
LIN {X 0,Y 425.28,Z 309.504,A -85,B 0,C 180,E1 20916.933,E2 20916.933} C_VEL
LIN {X 0,Y 425.281,Z 309.5,A -85,B 0,C 180,E1 20913.181,E2 20913.181} C_VEL
LIN {X 0,Y 425.298,Z 309.492,A -85,B 0,C 180,E1 20909.43,E2 20909.43} C_VEL
LIN {X 0,Y 425.31,Z 309.492,A -85,B 0,C 180,E1 20905.631,E2 20905.631} C_VEL
LIN {X 0,Y 425.32,Z 309.507,A -85,B 0,C 180,E1 20901.79,E2 20901.79} C_VEL
LIN {X 0,Y 425.296,Z 309.501,A -85,B 0,C 180,E1 20897.938,E2 20897.938} C_VEL
LIN {X 0,Y 425.262,Z 309.49,A -85,B 0,C 180,E1 20894.293,E2 20894.293} C_VEL
LIN {X 0,Y 425.254,Z 309.509,A -85,B 0,C 180,E1 20890.568,E2 20890.568} C_VEL
LIN {X 0,Y 425.25,Z 309.511,A -85,B 0,C 180,E1 20886.752,E2 20886.752} C_VEL
LIN {X 0,Y 425.262,Z 309.489,A -85,B 0,C 180,E1 20883.1,E2 20883.1} C_VEL
LIN {X 0,Y 425.286,Z 309.505,A -85,B 0,C 180,E1 20879.327,E2 20879.327} C_VEL
LIN {X 0,Y 425.292,Z 309.502,A -85,B 0,C 180,E1 20875.409,E2 20875.409} C_VEL
LIN {X 0,Y 425.286,Z 309.489,A -85,B 0,C 180,E1 20871.619,E2 20871.619} C_VEL
LIN {X 0,Y 425.266,Z 309.506,A -85,B 0,C 180,E1 20867.922,E2 20867.922} C_VEL
LIN {X 0,Y 425.258,Z 309.511,A -85,B 0,C 180,E1 20864.313,E2 20864.313} C_VEL
LIN {X 0,Y 425.265,Z 309.505,A -85,B 0,C 180,E1 20860.497,E2 20860.497} C_VEL
LIN {X 0,Y 425.282,Z 309.495,A -85,B 0,C 180,E1 20856.736,E2 20856.736} C_VEL
LIN {X 0,Y 425.308,Z 309.493,A -85,B 0,C 180,E1 20852.995,E2 20852.995} C_VEL
LIN {X 0,Y 425.323,Z 309.493,A -85,B 0,C 180,E1 20849.171,E2 20849.171} C_VEL
LIN {X 0,Y 425.308,Z 309.471,A -85,B 0,C 180,E1 20845.325,E2 20845.325} C_VEL
LIN {X 0,Y 425.306,Z 309.504,A -85,B 0,C 180,E1 20841.465,E2 20841.465} C_VEL
LIN {X 0,Y 425.285,Z 309.467,A -85,B 0,C 180,E1 20837.748,E2 20837.748} C_VEL
LIN {X 0,Y 425.365,Z 309.797,A -85,B 0,C 180,E1 20837.072,E2 20837.072} C_VEL
LIN {X 0,Y 426.875,Z 313.366,A -85,B 0,C 180,E1 20836.479,E2 20836.479} C_VEL
LIN {X 0,Y 435.021,Z 330.98,A -85,B 0,C 180,E1 20833.9,E2 20833.9} C_VEL
LIN {X 0,Y 442.907,Z 349.683,A -85,B 0,C 180,E1 20831.454,E2 20831.454} C_VEL
LIN {X 0,Y 446.657,Z 359.89,A -85,B 0,C 180,E1 20830.241,E2 20830.241} C_VEL
LIN {X 0,Y 444.624,Z 384.536,A -85,B 0,C 180,E1 20828.424,E2 20828.424} C_VEL
LIN {X 0,Y 448.182,Z 418.162,A -85,B 0,C 180,E1 20827.434,E2 20827.434} C_VEL
LIN {X 0,Y 442.654,Z 636.743,A -85,B 0,C 180,E1 20823.483,E2 20823.483} C_VEL
LIN {X 0,Y 441.487,Z 658.553,A -85,B 0,C 180,E1 20822.914,E2 20822.914} C_VEL
LIN {X 0,Y 439.862,Z 679.388,A -85,B 0,C 180,E1 20822.133,E2 20822.133} C_VEL
LIN {X 0,Y 438.112,Z 699.129,A -85,B 0,C 180,E1 20821.149,E2 20821.149} C_VEL
LIN {X 0,Y 436.149,Z 718.774,A -85,B 0,C 180,E1 20819.915,E2 20819.915} C_VEL
LIN {X 0,Y 434.065,Z 738.298,A -85,B 0,C 180,E1 20818.402,E2 20818.402} C_VEL
LIN {X 0,Y 432.059,Z 756.705,A -85,B 0,C 180,E1 20816.675,E2 20816.675} C_VEL
LIN {X 0,Y 430.138,Z 774.036,A -85,B 0,C 180,E1 20814.734,E2 20814.734} C_VEL
LIN {X 0,Y 428.44,Z 790.259,A -85,B 0,C 180,E1 20812.575,E2 20812.575} C_VEL
LIN {X 0,Y 427.035,Z 804.845,A -85,B 0,C 180,E1 20810.274,E2 20810.274} C_VEL
LIN {X 0,Y 425.959,Z 817.51,A -85,B 0,C 180,E1 20807.908,E2 20807.908} C_VEL
LIN {X 0,Y 425.186,Z 828.803,A -85,B 0,C 180,E1 20805.39,E2 20805.39} C_VEL
LIN {X 0,Y 424.667,Z 838.385,A -85,B 0,C 180,E1 20802.786,E2 20802.786} C_VEL
LIN {X 0,Y 424.416,Z 845.701,A -85,B 0,C 180,E1 20800.314,E2 20800.314} C_VEL
LIN {X 0,Y 424.309,Z 851.575,A -85,B 0,C 180,E1 20797.719,E2 20797.719} C_VEL
LIN {X 0,Y 424.311,Z 855.65,A -85,B 0,C 180,E1 20795.137,E2 20795.137} C_VEL
LIN {X 0,Y 424.338,Z 858.142,A -85,B 0,C 180,E1 20792.488,E2 20792.488} C_VEL
LIN {X 0,Y 424.358,Z 858.961,A -85,B 0,C 180,E1 20790,E2 20790} C_VEL
LIN {X 0,Y 424.339,Z 858.102,A -85,B 0,C 180,E1 20787.434,E2 20787.434} C_VEL
LIN {X 0,Y 424.311,Z 855.659,A -85,B 0,C 180,E1 20784.863,E2 20784.863} C_VEL
LIN {X 0,Y 424.308,Z 851.579,A -85,B 0,C 180,E1 20782.281,E2 20782.281} C_VEL
LIN {X 0,Y 424.417,Z 845.711,A -85,B 0,C 180,E1 20779.686,E2 20779.686} C_VEL
LIN {X 0,Y 424.667,Z 838.393,A -85,B 0,C 180,E1 20777.214,E2 20777.214} C_VEL
LIN {X 0,Y 425.192,Z 828.726,A -85,B 0,C 180,E1 20774.59,E2 20774.59} C_VEL
LIN {X 0,Y 425.959,Z 817.513,A -85,B 0,C 180,E1 20772.092,E2 20772.092} C_VEL
LIN {X 0,Y 427.036,Z 804.848,A -85,B 0,C 180,E1 20769.726,E2 20769.726} C_VEL
LIN {X 0,Y 428.441,Z 790.258,A -85,B 0,C 180,E1 20767.425,E2 20767.425} C_VEL
LIN {X 0,Y 430.138,Z 774.029,A -85,B 0,C 180,E1 20765.266,E2 20765.266} C_VEL
LIN {X 0,Y 432.059,Z 756.695,A -85,B 0,C 180,E1 20763.325,E2 20763.325} C_VEL
LIN {X 0,Y 434.064,Z 738.281,A -85,B 0,C 180,E1 20761.598,E2 20761.598} C_VEL
LIN {X 0,Y 436.146,Z 718.743,A -85,B 0,C 180,E1 20760.085,E2 20760.085} C_VEL
LIN {X 0,Y 438.106,Z 699.108,A -85,B 0,C 180,E1 20758.852,E2 20758.852} C_VEL
LIN {X 0,Y 439.858,Z 679.336,A -85,B 0,C 180,E1 20757.866,E2 20757.866} C_VEL
LIN {X 0,Y 441.493,Z 658.348,A -85,B 0,C 180,E1 20757.081,E2 20757.081} C_VEL
LIN {X 0,Y 442.667,Z 636.086,A -85,B 0,C 180,E1 20756.506,E2 20756.506} C_VEL
LIN {X 0,Y 448.204,Z 416.738,A -85,B 0,C 180,E1 20752.543,E2 20752.543} C_VEL
LIN {X 0,Y 444.573,Z 383.333,A -85,B 0,C 180,E1 20751.523,E2 20751.523} C_VEL
LIN {X 0,Y 446.59,Z 359.288,A -85,B 0,C 180,E1 20749.709,E2 20749.709} C_VEL
LIN {X 0,Y 438.573,Z 339.092,A -85,B 0,C 180,E1 20747.206,E2 20747.206} C_VEL
LIN {X 0,Y 430.583,Z 321.167,A -85,B 0,C 180,E1 20744.716,E2 20744.716} C_VEL
LIN {X 0,Y 425.441,Z 310.203,A -85,B 0,C 180,E1 20743.04,E2 20743.04} C_VEL
LIN {X 0,Y 425.323,Z 309.528,A -85,B 0,C 180,E1 20742.796,E2 20742.796} C_VEL
LIN {X 0,Y 425.328,Z 309.508,A -85,B 0,C 180,E1 20738.914,E2 20738.914} C_VEL
LIN {X 0,Y 425.312,Z 309.465,A -85,B 0,C 180,E1 20735.002,E2 20735.002} C_VEL
LIN {X 0,Y 425.293,Z 309.498,A -85,B 0,C 180,E1 20731.303,E2 20731.303} C_VEL
LIN {X 0,Y 425.275,Z 309.499,A -85,B 0,C 180,E1 20727.584,E2 20727.584} C_VEL
LIN {X 0,Y 425.269,Z 309.503,A -85,B 0,C 180,E1 20723.853,E2 20723.853} C_VEL
LIN {X 0,Y 425.274,Z 309.507,A -85,B 0,C 180,E1 20720.075,E2 20720.075} C_VEL
